	{attribute 'TcIecLibraryType'}
	{attribute 'external_name' := 'F_VN_HoughCircles_GUID_3208ACBE_0E75_B691_48A0_E9F1062BC23D'}
	(* Search for circles using the Hough transform. *)
	FUNCTION F_VN_HoughCircles : HRESULT
	VAR_INPUT
		ipSrcImage	:	ITcVnImage;	(* Source image (USINT, 1 channel, gray-level) *)
		ipCircles	:	REFERENCE TO ITcVnContainer;	(* Returns a container which is filled with the found circles (ContainerType_Vector_TcVnVector3_REAL; Each container element contains the x coordinate of the circle center [0], the y coordinate of the circle center [1], and the radius [2], respectively. Non-zero interface pointers are reused.) *)
		fInvAccuRatio	:	LREAL;	(* Inverted ratio of the accumulator size in relation to the source image's size (must be > 0. A value of 2 means that the size is halved in both directions.) *)
		fMinDist	:	LREAL;	(* Smallest allowed distance of two circles (must be > 0) *)
		hrPrev	:	HRESULT;	(* HRESULT indicating the result of previous operations (If SUCCEEDED(hrPrev) equals false, no operation is executed.) *)
	END_VAR

END_FUNCTION

// Functions/Image Analysis/Object Detection/F_VN_HoughCirclesExp

	{attribute 'TcIecLibraryType'}
	{attribute 'external_name' := 'F_VN_HoughCirclesExp_GUID_0524CE7C_E163_BD73_5710_38E608D89C08'}
	(* Search for circles using the Hough transform. (expert function) *)
	FUNCTION F_VN_HoughCirclesExp : HRESULT
	VAR_INPUT
		ipSrcImage	:	ITcVnImage;	(* Source image (USINT, 1 channel, gray-level) *)
		ipCircles	:	REFERENCE TO ITcVnContainer;	(* Returns a container which is filled with the found circles (ContainerType_Vector_TcVnVector3_REAL; Each container element contains the x coordinate of the circle center [0], the y coordinate of the circle center [1], and the radius [2], respectively. Non-zero interface pointers are reused.) *)
		fInvAccuRatio	:	LREAL;	(* Inverted ratio of the accumulator size in relation to the source image's size (must be > 0. A value of 2 means that the size is halved in both directions.) *)
		fMinDist	:	LREAL;	(* Smallest allowed distance of two circles (must be > 0) *)
		eHoughMethod	:	ETcVnHoughMethod;	(* Hough method to use (GRADIENT or GRADIENT_ALT) *)
		fParam1	:	LREAL;	(* First method specific parameter (GRADIENT, GRADIENT_ALT: upper threshold for canny edge detection, which must be > 0) *)
		fParam2	:	LREAL;	(* Second method specific parameter (GRADIENT: accumulator threshold for detecting circle centers, which must be > 0. GRADIENT_ALT: required circle perfectness, which must be > 0 and < 1, 1 would be a perfect circle) *)
		nMinRadius	:	UDINT;	(* Minimum circle radius allowed *)
		nMaxRadius	:	UDINT;	(* Maximum circle radius allowed (if 0, the value is internally set to max(image rows, image columns)) *)
		hrPrev	:	HRESULT;	(* HRESULT indicating the result of previous operations (If SUCCEEDED(hrPrev) equals false, no operation is executed.) *)
	END_VAR

END_FUNCTION

// Functions/Image Analysis/Object Detection/F_VN_HoughLines

	{attribute 'TcIecLibraryType'}
	{attribute 'external_name' := 'F_VN_HoughLines_GUID_82B94089_EA06_BA4D_5261_BCC69C56E98D'}
	(* Search for lines using the standard Hough transform. *)
	FUNCTION F_VN_HoughLines : HRESULT
	VAR_INPUT
		ipSrcImage	:	ITcVnImage;	(* Source image (USINT, 1 channel, binary, may be modified by the function) *)
		ipLines	:	REFERENCE TO ITcVnContainer;	(* Returns a container which is filled with the found lines (ContainerType_Vector_TcVnVector2_REAL; Each container element contains the distance from the origin [0] in pixels and the rotation angle [1] in radians, respectively. Non-zero interface pointers are reused.) *)
		fDistRes	:	LREAL;	(* Distance resolution of the accumulator (in pixels, must be > 0) *)
		fAngleRes	:	LREAL;	(* Angle resolution of the accumulator (in radians, must be > 0) *)
		nAccuThreshold	:	UDINT;	(* Accumulator threshold *)
		hrPrev	:	HRESULT;	(* HRESULT indicating the result of previous operations (If SUCCEEDED(hrPrev) equals false, no operation is executed.) *)
	END_VAR

END_FUNCTION

// Functions/Image Analysis/Object Detection/F_VN_HoughLinesExp

	{attribute 'TcIecLibraryType'}
	{attribute 'external_name' := 'F_VN_HoughLinesExp_GUID_A8676CC7_78FE_BBDF_4F0A_7E04EE46C3BD'}
	(* Search for lines using the standard Hough transform. (expert function) *)
	FUNCTION F_VN_HoughLinesExp : HRESULT
	VAR_INPUT
		ipSrcImage	:	ITcVnImage;	(* Source image (USINT, 1 channel, binary, may be modified by the function) *)
		ipLines	:	REFERENCE TO ITcVnContainer;	(* Returns a container which is filled with the found lines (ContainerType_Vector_TcVnVector2_REAL; Each container element contains the distance from the origin [0] in pixels and the rotation angle [1] in radians, respectively. Non-zero interface pointers are reused.) *)
		fDistRes	:	LREAL;	(* Distance resolution of the accumulator (in pixels, must be > 0) *)
		fAngleRes	:	LREAL;	(* Angle resolution of the accumulator (in radians, must be > 0) *)
		nAccuThreshold	:	UDINT;	(* Accumulator threshold *)
		fDistResDiv	:	LREAL;	(* Divisor of the distance resolution for the multi-scale Hough transform (>= 0, must be > 0 if fAngleResDiv is > 0) *)
		fAngleResDiv	:	LREAL;	(* Divisor of the angle resolution for the multi-scale Hough transform (>= 0, must be > 0 if fDistResDiv is > 0) *)
		hrPrev	:	HRESULT;	(* HRESULT indicating the result of previous operations (If SUCCEEDED(hrPrev) equals false, no operation is executed.) *)
	END_VAR

END_FUNCTION

// Functions/Image Analysis/Object Detection/F_VN_HoughLinesP

	{attribute 'TcIecLibraryType'}
	{attribute 'external_name' := 'F_VN_HoughLinesP_GUID_56A4DCAE_2908_B179_6CC2_F0080DB2F514'}
	(* Search for line segments using the probabilistic Hough transform. *)
	FUNCTION F_VN_HoughLinesP : HRESULT
	VAR_INPUT
		ipSrcImage	:	ITcVnImage;	(* Source image (USINT, 1 channel, binary, may be modified by the function) *)
		ipLines	:	REFERENCE TO ITcVnContainer;	(* Returns a container which is filled with the found line segments (ContainerType_Vector_TcVnVector4_DINT; Each container element contains the two ending points. Non-zero interface pointers are reused.) *)
		fDistRes	:	LREAL;	(* Distance resolution of the accumulator (in pixels, must be > 0) *)
		fAngleRes	:	LREAL;	(* Angle resolution of the accumulator (in radians, must be > 0) *)
		nAccuThreshold	:	UDINT;	(* Accumulator threshold *)
		hrPrev	:	HRESULT;	(* HRESULT indicating the result of previous operations (If SUCCEEDED(hrPrev) equals false, no operation is executed.) *)
	END_VAR

END_FUNCTION

// Functions/Image Analysis/Object Detection/F_VN_HoughLinesPExp

	{attribute 'TcIecLibraryType'}
	{attribute 'external_name' := 'F_VN_HoughLinesPExp_GUID_DBCDBAEB_C337_B034_483E_0DA75F1ED126'}
	(* Search for line segments using the probabilistic Hough transform. (expert function) *)
	FUNCTION F_VN_HoughLinesPExp : HRESULT
	VAR_INPUT
		ipSrcImage	:	ITcVnImage;	(* Source image (USINT, 1 channel, binary, may be modified by the function) *)
		ipLines	:	REFERENCE TO ITcVnContainer;	(* Returns a container which is filled with the found line segments (ContainerType_Vector_TcVnVector4_DINT; Each container element contains the two ending points. Non-zero interface pointers are reused.) *)
		fDistRes	:	LREAL;	(* Distance resolution of the accumulator (in pixels, must be > 0) *)
		fAngleRes	:	LREAL;	(* Angle resolution of the accumulator (in radians, must be > 0) *)
		nAccuThreshold	:	UDINT;	(* Accumulator threshold *)
		fMinLineLength	:	LREAL;	(* Minimum line length to search for *)
		fMaxLineGap	:	LREAL;	(* Maximum gap between points on the same line *)
		hrPrev	:	HRESULT;	(* HRESULT indicating the result of previous operations (If SUCCEEDED(hrPrev) equals false, no operation is executed.) *)
	END_VAR

END_FUNCTION

// Functions/Image Analysis/Object Detection/F_VN_MatchImageHuMoments

	{attribute 'TcIecLibraryType'}
	{attribute 'external_name' := 'F_VN_MatchImageHuMoments_GUID_658C7654_44DD_B199_410C_E15269A5A301'}
	(* Compare two images using the Hu moment invariants. *)
	FUNCTION F_VN_MatchImageHuMoments : HRESULT
	VAR_INPUT
		ipImage1	:	ITcVnImage;	(* First image (1 channel) *)
		ipImage2	:	ITcVnImage;	(* Second image (1 channel) *)
		eComparisonMethod	:	ETcVnContoursMatchComparisonMethod;	(* Method used for comparing the Hu moment invariants of the images *)
	END_VAR
	VAR_IN_OUT
		fDissimilarity	:	LREAL;	(* Returns the dissimilarity of the image Hu moment invariants depending on the chosen comparison method *)
	END_VAR
	VAR_INPUT
		hrPrev	:	HRESULT;	(* HRESULT indicating the result of previous operations (If SUCCEEDED(hrPrev) equals false, no operation is executed.) *)
	END_VAR

END_FUNCTION

// Functions/Image Analysis/Object Detection/F_VN_MatchTemplate

	{attribute 'TcIecLibraryType'}
	{attribute 'external_name' := 'F_VN_MatchTemplate_GUID_C0E3AE9A_E589_B4A4_40DE_437B35FB3E4E'}
	(* Match a template image with every location in the source image (using the TCVN_TMM_CCORR_NORMED method) and save the comparison results. *)
	FUNCTION F_VN_MatchTemplate : HRESULT
	VAR_INPUT
		ipSrcImage	:	ITcVnImage;	(* Source image (USINT or REAL, 1 or 3 channels) *)
		ipTemplateImage	:	ITcVnImage;	(* Template image (same type as ipSrcImage, smaller width and height) *)
		ipResultImage	:	REFERENCE TO ITcVnImage;	(* Returns the result image (REAL, normalized to [0..1], 1 channel, dimensions: (ipSrcImage.width - ipTemplateImage.width + 1) x (ipSrcImage.height - ipTemplateImage.height + 1). The best match is the global maximum. The position in ipResultImage is the top-left corner of ipTemplateImage position in ipSrcImage) *)
		hrPrev	:	HRESULT;	(* HRESULT indicating the result of previous operations (If SUCCEEDED(hrPrev) equals false, no operation is executed.) *)
	END_VAR

END_FUNCTION

// Functions/Image Analysis/Object Detection/F_VN_MatchTemplateExp

	{attribute 'TcIecLibraryType'}
	{attribute 'external_name' := 'F_VN_MatchTemplateExp_GUID_3688990C_CB5C_B619_7B29_C2927793ABF1'}
	(* Match a template image with every location in the source image and save the comparison results. (expert function) *)
	FUNCTION F_VN_MatchTemplateExp : HRESULT
	VAR_INPUT
		ipSrcImage	:	ITcVnImage;	(* Source image (USINT or REAL, 1 or 3 channels) *)
		ipTemplateImage	:	ITcVnImage;	(* Template image (same type as ipSrcImage, smaller width and height) *)
		ipResultImage	:	REFERENCE TO ITcVnImage;	(* Returns the result image (REAL, 1 channel, dimensions: (ipSrcImage.width - ipTemplateImage.width + 1) x (ipSrcImage.height - ipTemplateImage.height + 1). The best match is the global minimum (SQDIFF(_NORMED)) or maximum (CCORR(_NORMED), CCOEFF(_NORMED)). The position in ipResultImage is the top-left corner of ipTemplateImage position in ipSrcImage) *)
		eMatchMethod	:	ETcVnTemplateMatchMethod;	(* Specifies the template match method *)
		ipTemplateMask	:	ITcVnImage;	(* Optional mask for ipTemplateImage (same type and size as ipTemplateImage) *)
		hrPrev	:	HRESULT;	(* HRESULT indicating the result of previous operations (If SUCCEEDED(hrPrev) equals false, no operation is executed.) *)
	END_VAR

END_FUNCTION

// Functions/Image Analysis/Object Detection/F_VN_MatchTemplateAndEvaluate

	{attribute 'TcIecLibraryType'}
	{attribute 'external_name' := 'F_VN_MatchTemplateAndEvaluate_GUID_D49E239B_E98E_B6BB_418B_C7F76F8FBBDE'}
	(* Match a template image with every location in the source image (using the TCVN_TMM_CCORR_NORMED method) and evaluate the comparison results. Returns a sorted list of possible matches (best match first). *)
	FUNCTION F_VN_MatchTemplateAndEvaluate : HRESULT
	VAR_INPUT
		ipSrcImage	:	ITcVnImage;	(* Source image (USINT or REAL, 1 or 3 channels) *)
		ipTemplateImage	:	ITcVnImage;	(* Template image (same type as ipSrcImage, smaller width and height) *)
		ipMatches	:	REFERENCE TO ITcVnContainer;	(* Returns the matching positions (ContainerType_Vector_TcVnPoint2_DINT, where each element represents the top-left corner of ipTemplateImage) in ipSrcImage, sorted by relevance (best match first) *)
		fMatchThreshold	:	REAL;	(* Threshold to separate relevant from irrelevant matches (0..1, 1.0  would be a perfect match. To find a suitable value, you could evaluate some sample result images of F_VN_MatchTemplate.) *)
		hrPrev	:	HRESULT;	(* HRESULT indicating the result of previous operations (If SUCCEEDED(hrPrev) equals false, no operation is executed.) *)
	END_VAR

END_FUNCTION

// Functions/Image Analysis/Object Detection/F_VN_MatchTemplateAndEvaluateExp

	{attribute 'TcIecLibraryType'}
	{attribute 'external_name' := 'F_VN_MatchTemplateAndEvaluateExp_GUID_52774CC8_42BC_B4E1_7940_5C35FFE0176F'}
	(* Match a template image with every location in the source image and evaluate the comparison results. Returns a sorted list of possible matches (best match first). (expert function) *)
	FUNCTION F_VN_MatchTemplateAndEvaluateExp : HRESULT
	VAR_INPUT
		ipSrcImage	:	ITcVnImage;	(* Source image (USINT or REAL, 1 or 3 channels) *)
		ipTemplateImage	:	ITcVnImage;	(* Template image (same type as ipSrcImage, smaller width and height) *)
		ipMatches	:	REFERENCE TO ITcVnContainer;	(* Returns the matching positions (ContainerType_Vector_TcVnPoint2_DINT, where each element represents the top-left corner of ipTemplateImage) in ipSrcImage, sorted by relevance (best match first) *)
		fMatchThreshold	:	REAL;	(* Threshold to separate relevant from irrelevant matches (0..1 for NORMED methods, otherwise dependent on template size and content. To find a suitable value, you could evaluate some sample result images of F_VN_MatchTemplateExp.) *)
		eMatchMethod	:	ETcVnTemplateMatchMethod;	(* Specifies the template match method *)
		ipTemplateMask	:	ITcVnImage;	(* Optional mask for ipTemplateImage (same type and size as ipTemplateImage) *)
		fScaleFactor	:	REAL;	(* Factor (0..1] to reduce source and template image width and height for better performance (but less accuracy!) *)
		eInterpolationType	:	ETcVnInterpolationType;	(* Image resize interpolation type (only used if fScaleFactor != 1, TCVN_IT_BILINEAR recommended for most cases) *)
		ipMatchValues	:	REFERENCE TO ITcVnContainer;	(* Optionally returns the matching values (ContainerType_Vector_REAL, same size and sort order as ipMatches. Set to 0 if not required.) *)
		hrPrev	:	HRESULT;	(* HRESULT indicating the result of previous operations (If SUCCEEDED(hrPrev) equals false, no operation is executed.) *)
	END_VAR

END_FUNCTION

// Functions/Basic Container Operations/F_VN_AppendToContainer/F_VN_AppendToContainer_ITcVnContainer

	{attribute 'TcIecLibraryType'}
	{attribute 'external_name' := 'F_VN_AppendToContainer_ITcVnContainer_GUID_0871CEBE_66D6_B0B1_506F_1DCDB966BE0C'}
	(* Append a single element to a container or concatenate containers (if ipElement has the same typeId as ipContainer). *)
	FUNCTION F_VN_AppendToContainer_ITcVnContainer : HRESULT
	VAR_INPUT
		ipElement	:	ITcVnContainer;	(* Single element to append to ipContainer or container with several elements to be concatenated *)
		ipContainer	:	ITcVnContainer;	(* Container to which the element(s) will be appended *)
		hrPrev	:	HRESULT;	(* HRESULT indicating the result of previous operations (If SUCCEEDED(hrPrev) equals false, no operation is executed.) *)
	END_VAR

END_FUNCTION

// Functions/Basic Container Operations/F_VN_AppendToContainer/F_VN_AppendToContainer_ITcVnForwardIterator

	{attribute 'TcIecLibraryType'}
	{attribute 'external_name' := 'F_VN_AppendToContainer_ITcVnForwardIterator_GUID_68FE249C_FAB2_B211_7831_6890B9756309'}
	(* Append a single element (represented by an iterator)to a container. *)
	FUNCTION F_VN_AppendToContainer_ITcVnForwardIterator : HRESULT
	VAR_INPUT
		ipElement	:	ITcVnForwardIterator;	(* Single element to append to ipContainer *)
		ipContainer	:	ITcVnContainer;	(* Container to which the element(s) will be appended *)
		hrPrev	:	HRESULT;	(* HRESULT indicating the result of previous operations (If SUCCEEDED(hrPrev) equals false, no operation is executed.) *)
	END_VAR

END_FUNCTION

// Functions/Basic Container Operations/F_VN_AppendToContainer/F_VN_AppendToContainer_DINT

	{attribute 'TcIecLibraryType'}
	{attribute 'external_name' := 'F_VN_AppendToContainer_DINT_GUID_C5E3F485_1C44_B21C_61E3_958AE9652A0F'}
	(* Append a single element of type DINT to a container. *)
	FUNCTION F_VN_AppendToContainer_DINT : HRESULT
	VAR_INPUT
		nElement	:	DINT;	(* Single element to append to ipContainer *)
		ipContainer	:	ITcVnContainer;	(* Container to which the element will be appended *)
		hrPrev	:	HRESULT;	(* HRESULT indicating the result of previous operations (If SUCCEEDED(hrPrev) equals false, no operation is executed.) *)
	END_VAR

END_FUNCTION

// Functions/Basic Container Operations/F_VN_AppendToContainer/F_VN_AppendToContainer_INT

	{attribute 'TcIecLibraryType'}
	{attribute 'external_name' := 'F_VN_AppendToContainer_INT_GUID_1FA26B77_78C9_B37E_7C55_B9AB60A4781A'}
	(* Append a single element of type INT to a container. *)
	FUNCTION F_VN_AppendToContainer_INT : HRESULT
	VAR_INPUT
		nElement	:	INT;	(* Single element to append to ipContainer *)
		ipContainer	:	ITcVnContainer;	(* Container to which the element will be appended *)
		hrPrev	:	HRESULT;	(* HRESULT indicating the result of previous operations (If SUCCEEDED(hrPrev) equals false, no operation is executed.) *)
	END_VAR

END_FUNCTION

// Functions/Basic Container Operations/F_VN_AppendToContainer/F_VN_AppendToContainer_ITcVnImage

	{attribute 'TcIecLibraryType'}
	{attribute 'external_name' := 'F_VN_AppendToContainer_ITcVnImage_GUID_994AF0C6_0E53_B461_4DF2_1F839F8C5366'}
	(* Append a single element of type ITcVnImage to a container. *)
	FUNCTION F_VN_AppendToContainer_ITcVnImage : HRESULT
	VAR_INPUT
		ipElement	:	ITcVnImage;	(* Single element to append to ipContainer *)
		ipContainer	:	ITcVnContainer;	(* Container to which the element will be appended *)
		hrPrev	:	HRESULT;	(* HRESULT indicating the result of previous operations (If SUCCEEDED(hrPrev) equals false, no operation is executed.) *)
	END_VAR

END_FUNCTION

// Functions/Basic Container Operations/F_VN_AppendToContainer/F_VN_AppendToContainer_LREAL

	{attribute 'TcIecLibraryType'}
	{attribute 'external_name' := 'F_VN_AppendToContainer_LREAL_GUID_322EEAAD_BF59_BEC4_5462_10B3F9F43735'}
	(* Append a single element of type LREAL to a container. *)
	FUNCTION F_VN_AppendToContainer_LREAL : HRESULT
	VAR_INPUT
		fElement	:	LREAL;	(* Single element to append to ipContainer *)
		ipContainer	:	ITcVnContainer;	(* Container to which the element will be appended *)
		hrPrev	:	HRESULT;	(* HRESULT indicating the result of previous operations (If SUCCEEDED(hrPrev) equals false, no operation is executed.) *)
	END_VAR

END_FUNCTION

// Functions/Basic Container Operations/F_VN_AppendToContainer/F_VN_AppendToContainer_REAL

	{attribute 'TcIecLibraryType'}
	{attribute 'external_name' := 'F_VN_AppendToContainer_REAL_GUID_2B2B32F2_F49E_B830_4DE6_D5239ABAA89F'}
	(* Append a single element of type REAL to a container. *)
	FUNCTION F_VN_AppendToContainer_REAL : HRESULT
	VAR_INPUT
		fElement	:	REAL;	(* Single element to append to ipContainer *)
		ipContainer	:	ITcVnContainer;	(* Container to which the element will be appended *)
		hrPrev	:	HRESULT;	(* HRESULT indicating the result of previous operations (If SUCCEEDED(hrPrev) equals false, no operation is executed.) *)
	END_VAR

END_FUNCTION

// Functions/Basic Container Operations/F_VN_AppendToContainer/F_VN_AppendToContainer_SINT

	{attribute 'TcIecLibraryType'}
	{attribute 'external_name' := 'F_VN_AppendToContainer_SINT_GUID_AD0EA3F8_4615_B49A_4901_B8FA24011DED'}
	(* Append a single element of type SINT to a container. *)
	FUNCTION F_VN_AppendToContainer_SINT : HRESULT
	VAR_INPUT
		nElement	:	SINT;	(* Single element to append to ipContainer *)
		ipContainer	:	ITcVnContainer;	(* Container to which the element will be appended *)
		hrPrev	:	HRESULT;	(* HRESULT indicating the result of previous operations (If SUCCEEDED(hrPrev) equals false, no operation is executed.) *)
	END_VAR

END_FUNCTION

// Functions/Basic Container Operations/F_VN_AppendToContainer/F_VN_AppendToContainer_TcVnDMatch

	{attribute 'TcIecLibraryType'}
	{attribute 'external_name' := 'F_VN_AppendToContainer_TcVnDMatch_GUID_B7089787_0242_B315_4452_3A9278244513'}
	(* Append a single element of type TcVnDMatch to a container. *)
	FUNCTION F_VN_AppendToContainer_TcVnDMatch : HRESULT
	VAR_IN_OUT
		stElement	:	TcVnDMatch;	(* Single element to append to ipContainer *)
	END_VAR
	VAR_INPUT
		ipContainer	:	ITcVnContainer;	(* Container to which the element will be appended *)
		hrPrev	:	HRESULT;	(* HRESULT indicating the result of previous operations (If SUCCEEDED(hrPrev) equals false, no operation is executed.) *)
	END_VAR

END_FUNCTION

// Functions/Basic Container Operations/F_VN_AppendToContainer/F_VN_AppendToContainer_TcVnKeyPoint

	{attribute 'TcIecLibraryType'}
	{attribute 'external_name' := 'F_VN_AppendToContainer_TcVnKeyPoint_GUID_5E909463_2C7F_B636_51C1_80D41999F1FF'}
	(* Append a single element of type TcVnKeyPoint to a container. *)
	FUNCTION F_VN_AppendToContainer_TcVnKeyPoint : HRESULT
	VAR_IN_OUT
		stElement	:	TcVnKeyPoint;	(* Single element to append to ipContainer *)
	END_VAR
	VAR_INPUT
		ipContainer	:	ITcVnContainer;	(* Container to which the element will be appended *)
		hrPrev	:	HRESULT;	(* HRESULT indicating the result of previous operations (If SUCCEEDED(hrPrev) equals false, no operation is executed.) *)
	END_VAR

END_FUNCTION

// Functions/Basic Container Operations/F_VN_AppendToContainer/F_VN_AppendToContainer_TcVnPoint2_DINT

	{attribute 'TcIecLibraryType'}
	{attribute 'external_name' := 'F_VN_AppendToContainer_TcVnPoint2_DINT_GUID_61BA2EFB_B8BC_BFA0_630E_75DD36BF3AF5'}
	(* Append a single element of type TcVnPoint2_DINT to a container. *)
	FUNCTION F_VN_AppendToContainer_TcVnPoint2_DINT : HRESULT
	VAR_IN_OUT
		aElement	:	TcVnPoint2_DINT;	(* Single element to append to ipContainer *)
	END_VAR
	VAR_INPUT
		ipContainer	:	ITcVnContainer;	(* Container to which the element will be appended *)
		hrPrev	:	HRESULT;	(* HRESULT indicating the result of previous operations (If SUCCEEDED(hrPrev) equals false, no operation is executed.) *)
	END_VAR

END_FUNCTION

// Functions/Basic Container Operations/F_VN_AppendToContainer/F_VN_AppendToContainer_TcVnPoint2_LREAL

	{attribute 'TcIecLibraryType'}
	{attribute 'external_name' := 'F_VN_AppendToContainer_TcVnPoint2_LREAL_GUID_9578CCDD_C312_B676_7B95_A36643CB113E'}
	(* Append a single element of type TcVnPoint2_LREAL to a container. *)
	FUNCTION F_VN_AppendToContainer_TcVnPoint2_LREAL : HRESULT
	VAR_IN_OUT
		aElement	:	TcVnPoint2_LREAL;	(* Single element to append to ipContainer *)
	END_VAR
	VAR_INPUT
		ipContainer	:	ITcVnContainer;	(* Container to which the element will be appended *)
		hrPrev	:	HRESULT;	(* HRESULT indicating the result of previous operations (If SUCCEEDED(hrPrev) equals false, no operation is executed.) *)
	END_VAR

END_FUNCTION

// Functions/Basic Container Operations/F_VN_AppendToContainer/F_VN_AppendToContainer_TcVnPoint2_REAL

	{attribute 'TcIecLibraryType'}
	{attribute 'external_name' := 'F_VN_AppendToContainer_TcVnPoint2_REAL_GUID_2CACAC7F_BF8B_B238_50E3_05B26FF81174'}
	(* Append a single element of type TcVnPoint2_REAL to a container. *)
	FUNCTION F_VN_AppendToContainer_TcVnPoint2_REAL : HRESULT
	VAR_IN_OUT
		aElement	:	TcVnPoint2_REAL;	(* Single element to append to ipContainer *)
	END_VAR
	VAR_INPUT
		ipContainer	:	ITcVnContainer;	(* Container to which the element will be appended *)
		hrPrev	:	HRESULT;	(* HRESULT indicating the result of previous operations (If SUCCEEDED(hrPrev) equals false, no operation is executed.) *)
	END_VAR

END_FUNCTION

// Functions/Basic Container Operations/F_VN_AppendToContainer/F_VN_AppendToContainer_TcVnPoint3_LREAL

	{attribute 'TcIecLibraryType'}
	{attribute 'external_name' := 'F_VN_AppendToContainer_TcVnPoint3_LREAL_GUID_C00DAD65_4FEA_B107_711B_0C106CCBB85A'}
	(* Append a single element of type TcVnPoint3_LREAL to a container. *)
	FUNCTION F_VN_AppendToContainer_TcVnPoint3_LREAL : HRESULT
	VAR_IN_OUT
		aElement	:	TcVnPoint3_LREAL;	(* Single element to append to ipContainer *)
	END_VAR
	VAR_INPUT
		ipContainer	:	ITcVnContainer;	(* Container to which the element will be appended *)
		hrPrev	:	HRESULT;	(* HRESULT indicating the result of previous operations (If SUCCEEDED(hrPrev) equals false, no operation is executed.) *)
	END_VAR

END_FUNCTION

// Functions/Basic Container Operations/F_VN_AppendToContainer/F_VN_AppendToContainer_TcVnPoint3_REAL

	{attribute 'TcIecLibraryType'}
	{attribute 'external_name' := 'F_VN_AppendToContainer_TcVnPoint3_REAL_GUID_DCD53F51_0FDB_B6B9_6DCB_4B5117963B6D'}
	(* Append a single element of type TcVnPoint3_REAL to a container. *)
	FUNCTION F_VN_AppendToContainer_TcVnPoint3_REAL : HRESULT
	VAR_IN_OUT
		aElement	:	TcVnPoint3_REAL;	(* Single element to append to ipContainer *)
	END_VAR
	VAR_INPUT
		ipContainer	:	ITcVnContainer;	(* Container to which the element will be appended *)
		hrPrev	:	HRESULT;	(* HRESULT indicating the result of previous operations (If SUCCEEDED(hrPrev) equals false, no operation is executed.) *)
	END_VAR

END_FUNCTION

// Functions/Basic Container Operations/F_VN_AppendToContainer/F_VN_AppendToContainer_TcVnRectangle_DINT

	{attribute 'TcIecLibraryType'}
	{attribute 'external_name' := 'F_VN_AppendToContainer_TcVnRectangle_DINT_GUID_C4A818BF_201D_B4FB_7B4B_564F3F6D47CE'}
	(* Append a single element of type TcVnRectangle_DINT to a container. *)
	FUNCTION F_VN_AppendToContainer_TcVnRectangle_DINT : HRESULT
	VAR_IN_OUT
		stElement	:	TcVnRectangle_DINT;	(* Single element to append to ipContainer *)
	END_VAR
	VAR_INPUT
		ipContainer	:	ITcVnContainer;	(* Container to which the element will be appended *)
		hrPrev	:	HRESULT;	(* HRESULT indicating the result of previous operations (If SUCCEEDED(hrPrev) equals false, no operation is executed.) *)
	END_VAR

END_FUNCTION

// Functions/Basic Container Operations/F_VN_AppendToContainer/F_VN_AppendToContainer_TcVnVector2_DINT

	{attribute 'TcIecLibraryType'}
	{attribute 'external_name' := 'F_VN_AppendToContainer_TcVnVector2_DINT_GUID_41B34E71_A627_B579_4E88_D7D74BBEB1E5'}
	(* Append a single element of type TcVnVector2_DINT to a container. *)
	FUNCTION F_VN_AppendToContainer_TcVnVector2_DINT : HRESULT
	VAR_IN_OUT
		aElement	:	TcVnVector2_DINT;	(* Single element to append to ipContainer *)
	END_VAR
	VAR_INPUT
		ipContainer	:	ITcVnContainer;	(* Container to which the element will be appended *)
		hrPrev	:	HRESULT;	(* HRESULT indicating the result of previous operations (If SUCCEEDED(hrPrev) equals false, no operation is executed.) *)
	END_VAR

END_FUNCTION

// Functions/Basic Container Operations/F_VN_AppendToContainer/F_VN_AppendToContainer_TcVnVector2_INT

	{attribute 'TcIecLibraryType'}
	{attribute 'external_name' := 'F_VN_AppendToContainer_TcVnVector2_INT_GUID_03190075_1655_BB8D_5670_7DFA56918C83'}
	(* Append a single element of type TcVnVector2_INT to a container. *)
	FUNCTION F_VN_AppendToContainer_TcVnVector2_INT : HRESULT
	VAR_IN_OUT
		aElement	:	TcVnVector2_INT;	(* Single element to append to ipContainer *)
	END_VAR
	VAR_INPUT
		ipContainer	:	ITcVnContainer;	(* Container to which the element will be appended *)
		hrPrev	:	HRESULT;	(* HRESULT indicating the result of previous operations (If SUCCEEDED(hrPrev) equals false, no operation is executed.) *)
	END_VAR

END_FUNCTION

// Functions/Basic Container Operations/F_VN_AppendToContainer/F_VN_AppendToContainer_TcVnVector2_REAL

	{attribute 'TcIecLibraryType'}
	{attribute 'external_name' := 'F_VN_AppendToContainer_TcVnVector2_REAL_GUID_CAA9172F_D581_B4EB_508B_C992A7AC72E9'}
	(* Append a single element of type TcVnVector2_REAL to a container. *)
	FUNCTION F_VN_AppendToContainer_TcVnVector2_REAL : HRESULT
	VAR_IN_OUT
		aElement	:	TcVnVector2_REAL;	(* Single element to append to ipContainer *)
	END_VAR
	VAR_INPUT
		ipContainer	:	ITcVnContainer;	(* Container to which the element will be appended *)
		hrPrev	:	HRESULT;	(* HRESULT indicating the result of previous operations (If SUCCEEDED(hrPrev) equals false, no operation is executed.) *)
	END_VAR

END_FUNCTION

// Functions/Basic Container Operations/F_VN_AppendToContainer/F_VN_AppendToContainer_TcVnVector2_SINT

	{attribute 'TcIecLibraryType'}
	{attribute 'external_name' := 'F_VN_AppendToContainer_TcVnVector2_SINT_GUID_B243487F_92C1_BF7E_71E2_97E88C51A164'}
	(* Append a single element of type TcVnVector2_SINT to a container. *)
	FUNCTION F_VN_AppendToContainer_TcVnVector2_SINT : HRESULT
	VAR_IN_OUT
		aElement	:	TcVnVector2_SINT;	(* Single element to append to ipContainer *)
	END_VAR
	VAR_INPUT
		ipContainer	:	ITcVnContainer;	(* Container to which the element will be appended *)
		hrPrev	:	HRESULT;	(* HRESULT indicating the result of previous operations (If SUCCEEDED(hrPrev) equals false, no operation is executed.) *)
	END_VAR

END_FUNCTION

// Functions/Basic Container Operations/F_VN_AppendToContainer/F_VN_AppendToContainer_TcVnVector2_UINT

	{attribute 'TcIecLibraryType'}
	{attribute 'external_name' := 'F_VN_AppendToContainer_TcVnVector2_UINT_GUID_65CA8312_34CD_BCB3_4316_349611E62963'}
	(* Append a single element of type TcVnVector2_UINT to a container. *)
	FUNCTION F_VN_AppendToContainer_TcVnVector2_UINT : HRESULT
	VAR_IN_OUT
		aElement	:	TcVnVector2_UINT;	(* Single element to append to ipContainer *)
	END_VAR
	VAR_INPUT
		ipContainer	:	ITcVnContainer;	(* Container to which the element will be appended *)
		hrPrev	:	HRESULT;	(* HRESULT indicating the result of previous operations (If SUCCEEDED(hrPrev) equals false, no operation is executed.) *)
	END_VAR

END_FUNCTION

// Functions/Basic Container Operations/F_VN_AppendToContainer/F_VN_AppendToContainer_TcVnVector2_USINT

	{attribute 'TcIecLibraryType'}
	{attribute 'external_name' := 'F_VN_AppendToContainer_TcVnVector2_USINT_GUID_CFDE5759_AA22_BAFD_4045_17761752DF7A'}
	(* Append a single element of type TcVnVector2_USINT to a container. *)
	FUNCTION F_VN_AppendToContainer_TcVnVector2_USINT : HRESULT
	VAR_IN_OUT
		aElement	:	TcVnVector2_USINT;	(* Single element to append to ipContainer *)
	END_VAR
	VAR_INPUT
		ipContainer	:	ITcVnContainer;	(* Container to which the element will be appended *)
		hrPrev	:	HRESULT;	(* HRESULT indicating the result of previous operations (If SUCCEEDED(hrPrev) equals false, no operation is executed.) *)
	END_VAR

END_FUNCTION

// Functions/Basic Container Operations/F_VN_AppendToContainer/F_VN_AppendToContainer_TcVnVector3_INT

	{attribute 'TcIecLibraryType'}
	{attribute 'external_name' := 'F_VN_AppendToContainer_TcVnVector3_INT_GUID_865E49A2_C2A9_B29E_4549_0BC3152D1033'}
	(* Append a single element of type TcVnVector3_INT to a container. *)
	FUNCTION F_VN_AppendToContainer_TcVnVector3_INT : HRESULT
	VAR_IN_OUT
		aElement	:	TcVnVector3_INT;	(* Single element to append to ipContainer *)
	END_VAR
	VAR_INPUT
		ipContainer	:	ITcVnContainer;	(* Container to which the element will be appended *)
		hrPrev	:	HRESULT;	(* HRESULT indicating the result of previous operations (If SUCCEEDED(hrPrev) equals false, no operation is executed.) *)
	END_VAR

END_FUNCTION

// Functions/Basic Container Operations/F_VN_AppendToContainer/F_VN_AppendToContainer_TcVnVector3_REAL

	{attribute 'TcIecLibraryType'}
	{attribute 'external_name' := 'F_VN_AppendToContainer_TcVnVector3_REAL_GUID_D2CCFE6F_59DD_B2C5_60F3_EB5A1DCAE86F'}
	(* Append a single element of type TcVnVector3_REAL to a container. *)
	FUNCTION F_VN_AppendToContainer_TcVnVector3_REAL : HRESULT
	VAR_IN_OUT
		aElement	:	TcVnVector3_REAL;	(* Single element to append to ipContainer *)
	END_VAR
	VAR_INPUT
		ipContainer	:	ITcVnContainer;	(* Container to which the element will be appended *)
		hrPrev	:	HRESULT;	(* HRESULT indicating the result of previous operations (If SUCCEEDED(hrPrev) equals false, no operation is executed.) *)
	END_VAR

END_FUNCTION

// Functions/Basic Container Operations/F_VN_AppendToContainer/F_VN_AppendToContainer_TcVnVector3_SINT

	{attribute 'TcIecLibraryType'}
	{attribute 'external_name' := 'F_VN_AppendToContainer_TcVnVector3_SINT_GUID_C0B410A5_2EC6_B0F0_49B3_B07241C8F6DE'}
	(* Append a single element of type TcVnVector3_SINT to a container. *)
	FUNCTION F_VN_AppendToContainer_TcVnVector3_SINT : HRESULT
	VAR_IN_OUT
		aElement	:	TcVnVector3_SINT;	(* Single element to append to ipContainer *)
	END_VAR
	VAR_INPUT
		ipContainer	:	ITcVnContainer;	(* Container to which the element will be appended *)
		hrPrev	:	HRESULT;	(* HRESULT indicating the result of previous operations (If SUCCEEDED(hrPrev) equals false, no operation is executed.) *)
	END_VAR

END_FUNCTION

// Functions/Basic Container Operations/F_VN_AppendToContainer/F_VN_AppendToContainer_TcVnVector3_UINT

	{attribute 'TcIecLibraryType'}
	{attribute 'external_name' := 'F_VN_AppendToContainer_TcVnVector3_UINT_GUID_F6024E8E_E5FB_BD9D_7C19_F5DA416AACF1'}
	(* Append a single element of type TcVnVector3_UINT to a container. *)
	FUNCTION F_VN_AppendToContainer_TcVnVector3_UINT : HRESULT
	VAR_IN_OUT
		aElement	:	TcVnVector3_UINT;	(* Single element to append to ipContainer *)
	END_VAR
	VAR_INPUT
		ipContainer	:	ITcVnContainer;	(* Container to which the element will be appended *)
		hrPrev	:	HRESULT;	(* HRESULT indicating the result of previous operations (If SUCCEEDED(hrPrev) equals false, no operation is executed.) *)
	END_VAR

END_FUNCTION

// Functions/Basic Container Operations/F_VN_AppendToContainer/F_VN_AppendToContainer_TcVnVector3_USINT

	{attribute 'TcIecLibraryType'}
	{attribute 'external_name' := 'F_VN_AppendToContainer_TcVnVector3_USINT_GUID_8B62F65E_08EA_B240_504E_B61CBAA0D91D'}
	(* Append a single element of type TcVnVector3_USINT to a container. *)
	FUNCTION F_VN_AppendToContainer_TcVnVector3_USINT : HRESULT
	VAR_IN_OUT
		aElement	:	TcVnVector3_USINT;	(* Single element to append to ipContainer *)
	END_VAR
	VAR_INPUT
		ipContainer	:	ITcVnContainer;	(* Container to which the element will be appended *)
		hrPrev	:	HRESULT;	(* HRESULT indicating the result of previous operations (If SUCCEEDED(hrPrev) equals false, no operation is executed.) *)
	END_VAR

END_FUNCTION

// Functions/Basic Container Operations/F_VN_AppendToContainer/F_VN_AppendToContainer_TcVnVector4_DINT

	{attribute 'TcIecLibraryType'}
	{attribute 'external_name' := 'F_VN_AppendToContainer_TcVnVector4_DINT_GUID_8BB3E3FF_2F4E_BC73_4B23_6733ABEE0780'}
	(* Append a single element of type TcVnVector4_DINT to a container. *)
	FUNCTION F_VN_AppendToContainer_TcVnVector4_DINT : HRESULT
	VAR_IN_OUT
		aElement	:	TcVnVector4_DINT;	(* Single element to append to ipContainer *)
	END_VAR
	VAR_INPUT
		ipContainer	:	ITcVnContainer;	(* Container to which the element will be appended *)
		hrPrev	:	HRESULT;	(* HRESULT indicating the result of previous operations (If SUCCEEDED(hrPrev) equals false, no operation is executed.) *)
	END_VAR

END_FUNCTION

// Functions/Basic Container Operations/F_VN_AppendToContainer/F_VN_AppendToContainer_TcVnVector4_INT

	{attribute 'TcIecLibraryType'}
	{attribute 'external_name' := 'F_VN_AppendToContainer_TcVnVector4_INT_GUID_80AE1EA5_7A7E_B9B0_4985_BB5D32954B0E'}
	(* Append a single element of type TcVnVector4_INT to a container. *)
	FUNCTION F_VN_AppendToContainer_TcVnVector4_INT : HRESULT
	VAR_IN_OUT
		aElement	:	TcVnVector4_INT;	(* Single element to append to ipContainer *)
	END_VAR
	VAR_INPUT
		ipContainer	:	ITcVnContainer;	(* Container to which the element will be appended *)
		hrPrev	:	HRESULT;	(* HRESULT indicating the result of previous operations (If SUCCEEDED(hrPrev) equals false, no operation is executed.) *)
	END_VAR

END_FUNCTION

// Functions/Basic Container Operations/F_VN_AppendToContainer/F_VN_AppendToContainer_TcVnVector4_LREAL

	{attribute 'TcIecLibraryType'}
	{attribute 'external_name' := 'F_VN_AppendToContainer_TcVnVector4_LREAL_GUID_EB913DE2_DA93_BA7B_473D_8239404B5042'}
	(* Append a single element of type TcVnVector4_LREAL to a container. *)
	FUNCTION F_VN_AppendToContainer_TcVnVector4_LREAL : HRESULT
	VAR_IN_OUT
		aElement	:	TcVnVector4_LREAL;	(* Single element to append to ipContainer *)
	END_VAR
	VAR_INPUT
		ipContainer	:	ITcVnContainer;	(* Container to which the element will be appended *)
		hrPrev	:	HRESULT;	(* HRESULT indicating the result of previous operations (If SUCCEEDED(hrPrev) equals false, no operation is executed.) *)
	END_VAR

END_FUNCTION

// Functions/Basic Container Operations/F_VN_AppendToContainer/F_VN_AppendToContainer_TcVnVector4_SINT

	{attribute 'TcIecLibraryType'}
	{attribute 'external_name' := 'F_VN_AppendToContainer_TcVnVector4_SINT_GUID_0C452B4A_D316_B59E_437F_F319934F215D'}
	(* Append a single element of type TcVnVector4_SINT to a container. *)
	FUNCTION F_VN_AppendToContainer_TcVnVector4_SINT : HRESULT
	VAR_IN_OUT
		aElement	:	TcVnVector4_SINT;	(* Single element to append to ipContainer *)
	END_VAR
	VAR_INPUT
		ipContainer	:	ITcVnContainer;	(* Container to which the element will be appended *)
		hrPrev	:	HRESULT;	(* HRESULT indicating the result of previous operations (If SUCCEEDED(hrPrev) equals false, no operation is executed.) *)
	END_VAR

END_FUNCTION

// Functions/Basic Container Operations/F_VN_AppendToContainer/F_VN_AppendToContainer_TcVnVector4_UINT

	{attribute 'TcIecLibraryType'}
	{attribute 'external_name' := 'F_VN_AppendToContainer_TcVnVector4_UINT_GUID_0032CD21_D254_B26C_7A07_E6D6874AB4CC'}
	(* Append a single element of type TcVnVector4_UINT to a container. *)
	FUNCTION F_VN_AppendToContainer_TcVnVector4_UINT : HRESULT
	VAR_IN_OUT
		aElement	:	TcVnVector4_UINT;	(* Single element to append to ipContainer *)
	END_VAR
	VAR_INPUT
		ipContainer	:	ITcVnContainer;	(* Container to which the element will be appended *)
		hrPrev	:	HRESULT;	(* HRESULT indicating the result of previous operations (If SUCCEEDED(hrPrev) equals false, no operation is executed.) *)
	END_VAR

END_FUNCTION

// Functions/Basic Container Operations/F_VN_AppendToContainer/F_VN_AppendToContainer_TcVnVector4_USINT

	{attribute 'TcIecLibraryType'}
	{attribute 'external_name' := 'F_VN_AppendToContainer_TcVnVector4_USINT_GUID_EC0B014C_363A_BF2F_6D81_097AF29A2E32'}
	(* Append a single element of type TcVnVector4_USINT to a container. *)
	FUNCTION F_VN_AppendToContainer_TcVnVector4_USINT : HRESULT
	VAR_IN_OUT
		aElement	:	TcVnVector4_USINT;	(* Single element to append to ipContainer *)
	END_VAR
	VAR_INPUT
		ipContainer	:	ITcVnContainer;	(* Container to which the element will be appended *)
		hrPrev	:	HRESULT;	(* HRESULT indicating the result of previous operations (If SUCCEEDED(hrPrev) equals false, no operation is executed.) *)
	END_VAR

END_FUNCTION

// Functions/Basic Container Operations/F_VN_AppendToContainer/F_VN_AppendToContainer_UDINT

	{attribute 'TcIecLibraryType'}
	{attribute 'external_name' := 'F_VN_AppendToContainer_UDINT_GUID_07FC158B_CFC8_B0A5_770B_691D25F2923E'}
	(* Append a single element of type UDINT to a container. *)
	FUNCTION F_VN_AppendToContainer_UDINT : HRESULT
	VAR_INPUT
		nElement	:	UDINT;	(* Single element to append to ipContainer *)
		ipContainer	:	ITcVnContainer;	(* Container to which the element will be appended *)
		hrPrev	:	HRESULT;	(* HRESULT indicating the result of previous operations (If SUCCEEDED(hrPrev) equals false, no operation is executed.) *)
	END_VAR

END_FUNCTION

// Functions/Basic Container Operations/F_VN_AppendToContainer/F_VN_AppendToContainer_UINT

	{attribute 'TcIecLibraryType'}
	{attribute 'external_name' := 'F_VN_AppendToContainer_UINT_GUID_BDB75763_84AF_B740_41A9_314125C5A350'}
	(* Append a single element of type UINT to a container. *)
	FUNCTION F_VN_AppendToContainer_UINT : HRESULT
	VAR_INPUT
		nElement	:	UINT;	(* Single element to append to ipContainer *)
		ipContainer	:	ITcVnContainer;	(* Container to which the element will be appended *)
		hrPrev	:	HRESULT;	(* HRESULT indicating the result of previous operations (If SUCCEEDED(hrPrev) equals false, no operation is executed.) *)
	END_VAR

END_FUNCTION

// Functions/Basic Container Operations/F_VN_AppendToContainer/F_VN_AppendToContainer_ULINT

	{attribute 'TcIecLibraryType'}
	{attribute 'external_name' := 'F_VN_AppendToContainer_ULINT_GUID_31AA49B0_A8DE_B40B_4286_64C865B39163'}
	(* Append a single element of type ULINT to a container. *)
	FUNCTION F_VN_AppendToContainer_ULINT : HRESULT
	VAR_INPUT
		nElement	:	ULINT;	(* Single element to append to ipContainer *)
		ipContainer	:	ITcVnContainer;	(* Container to which the element will be appended *)
		hrPrev	:	HRESULT;	(* HRESULT indicating the result of previous operations (If SUCCEEDED(hrPrev) equals false, no operation is executed.) *)
	END_VAR

END_FUNCTION

// Functions/Basic Container Operations/F_VN_AppendToContainer/F_VN_AppendToContainer_USINT

	{attribute 'TcIecLibraryType'}
	{attribute 'external_name' := 'F_VN_AppendToContainer_USINT_GUID_8F2D6821_4D5B_B313_5DEE_BB4B65282616'}
	(* Append a single element of type USINT to a container. *)
	FUNCTION F_VN_AppendToContainer_USINT : HRESULT
	VAR_INPUT
		nElement	:	USINT;	(* Single element to append to ipContainer *)
		ipContainer	:	ITcVnContainer;	(* Container to which the element will be appended *)
		hrPrev	:	HRESULT;	(* HRESULT indicating the result of previous operations (If SUCCEEDED(hrPrev) equals false, no operation is executed.) *)
	END_VAR

END_FUNCTION

// Functions/Basic Container Operations/F_VN_FillContainer/F_VN_FillContainer_DINT

	{attribute 'TcIecLibraryType'}
	{attribute 'external_name' := 'F_VN_FillContainer_DINT_GUID_8BB266DC_9DD3_B627_565F_7067D41D7538'}
	(* Fill the container with the specified value. Only possible for containers with basic elements. *)
	FUNCTION F_VN_FillContainer_DINT : HRESULT
	VAR_INPUT
		ipContainer	:	ITcVnContainer;	(* Container with basic elements *)
		nValue	:	DINT;	(* Value to set the container elements *)
		hrPrev	:	HRESULT;	(* HRESULT indicating the result of previous operations (If SUCCEEDED(hrPrev) equals false, no operation is executed.) *)
	END_VAR

END_FUNCTION

// Functions/Basic Container Operations/F_VN_FillContainer/F_VN_FillContainer_INT

	{attribute 'TcIecLibraryType'}
	{attribute 'external_name' := 'F_VN_FillContainer_INT_GUID_0D5FEBDD_6399_B344_4F23_559608459CC7'}
	(* Fill the container with the specified value. Only possible for containers with basic elements. *)
	FUNCTION F_VN_FillContainer_INT : HRESULT
	VAR_INPUT
		ipContainer	:	ITcVnContainer;	(* Container with basic elements *)
		nValue	:	INT;	(* Value to set the container elements *)
		hrPrev	:	HRESULT;	(* HRESULT indicating the result of previous operations (If SUCCEEDED(hrPrev) equals false, no operation is executed.) *)
	END_VAR

END_FUNCTION

// Functions/Basic Container Operations/F_VN_FillContainer/F_VN_FillContainer_ITcVnImage

	{attribute 'TcIecLibraryType'}
	{attribute 'external_name' := 'F_VN_FillContainer_ITcVnImage_GUID_A1258E31_3B81_BA73_614D_90858A512D0D'}
	(* Fill the container with the specified value. Only possible for containers with basic elements. *)
	FUNCTION F_VN_FillContainer_ITcVnImage : HRESULT
	VAR_INPUT
		ipContainer	:	ITcVnContainer;	(* Container with basic elements *)
		ipValue	:	ITcVnImage;	(* Value to set the container elements *)
		hrPrev	:	HRESULT;	(* HRESULT indicating the result of previous operations (If SUCCEEDED(hrPrev) equals false, no operation is executed.) *)
	END_VAR

END_FUNCTION

// Functions/Basic Container Operations/F_VN_FillContainer/F_VN_FillContainer_LREAL

	{attribute 'TcIecLibraryType'}
	{attribute 'external_name' := 'F_VN_FillContainer_LREAL_GUID_0EB3FA1D_6B4E_B9F9_57FC_0DED14EB922F'}
	(* Fill the container with the specified value. Only possible for containers with basic elements. *)
	FUNCTION F_VN_FillContainer_LREAL : HRESULT
	VAR_INPUT
		ipContainer	:	ITcVnContainer;	(* Container with basic elements *)
		fValue	:	LREAL;	(* Value to set the container elements *)
		hrPrev	:	HRESULT;	(* HRESULT indicating the result of previous operations (If SUCCEEDED(hrPrev) equals false, no operation is executed.) *)
	END_VAR

END_FUNCTION

// Functions/Basic Container Operations/F_VN_FillContainer/F_VN_FillContainer_REAL

	{attribute 'TcIecLibraryType'}
	{attribute 'external_name' := 'F_VN_FillContainer_REAL_GUID_53B9D44F_7269_B320_6944_9E8CB7215B15'}
	(* Fill the container with the specified value. Only possible for containers with basic elements. *)
	FUNCTION F_VN_FillContainer_REAL : HRESULT
	VAR_INPUT
		ipContainer	:	ITcVnContainer;	(* Container with basic elements *)
		fValue	:	REAL;	(* Value to set the container elements *)
		hrPrev	:	HRESULT;	(* HRESULT indicating the result of previous operations (If SUCCEEDED(hrPrev) equals false, no operation is executed.) *)
	END_VAR

END_FUNCTION

// Functions/Basic Container Operations/F_VN_FillContainer/F_VN_FillContainer_SINT

	{attribute 'TcIecLibraryType'}
	{attribute 'external_name' := 'F_VN_FillContainer_SINT_GUID_74859358_058A_B104_5BCB_AD33D56BA120'}
	(* Fill the container with the specified value. Only possible for containers with basic elements. *)
	FUNCTION F_VN_FillContainer_SINT : HRESULT
	VAR_INPUT
		ipContainer	:	ITcVnContainer;	(* Container with basic elements *)
		nValue	:	SINT;	(* Value to set the container elements *)
		hrPrev	:	HRESULT;	(* HRESULT indicating the result of previous operations (If SUCCEEDED(hrPrev) equals false, no operation is executed.) *)
	END_VAR

END_FUNCTION

// Functions/Basic Container Operations/F_VN_FillContainer/F_VN_FillContainer_TcVnDMatch

	{attribute 'TcIecLibraryType'}
	{attribute 'external_name' := 'F_VN_FillContainer_TcVnDMatch_GUID_1945276A_7A89_B552_5CEE_6CF2E817D3E8'}
	(* Fill the container with the specified value. Only possible for containers with basic elements. *)
	FUNCTION F_VN_FillContainer_TcVnDMatch : HRESULT
	VAR_INPUT
		ipContainer	:	ITcVnContainer;	(* Container with basic elements *)
	END_VAR
	VAR_IN_OUT
		stValue	:	TcVnDMatch;	(* Value to set the container elements *)
	END_VAR
	VAR_INPUT
		hrPrev	:	HRESULT;	(* HRESULT indicating the result of previous operations (If SUCCEEDED(hrPrev) equals false, no operation is executed.) *)
	END_VAR

END_FUNCTION

// Functions/Basic Container Operations/F_VN_FillContainer/F_VN_FillContainer_TcVnKeyPoint

	{attribute 'TcIecLibraryType'}
	{attribute 'external_name' := 'F_VN_FillContainer_TcVnKeyPoint_GUID_93F5697E_0406_B001_550F_074DFB818BFF'}
	(* Fill the container with the specified value. Only possible for containers with basic elements. *)
	FUNCTION F_VN_FillContainer_TcVnKeyPoint : HRESULT
	VAR_INPUT
		ipContainer	:	ITcVnContainer;	(* Container with basic elements *)
	END_VAR
	VAR_IN_OUT
		stValue	:	TcVnKeyPoint;	(* Value to set the container elements *)
	END_VAR
	VAR_INPUT
		hrPrev	:	HRESULT;	(* HRESULT indicating the result of previous operations (If SUCCEEDED(hrPrev) equals false, no operation is executed.) *)
	END_VAR

END_FUNCTION

// Functions/Basic Container Operations/F_VN_FillContainer/F_VN_FillContainer_TcVnPoint2_DINT

	{attribute 'TcIecLibraryType'}
	{attribute 'external_name' := 'F_VN_FillContainer_TcVnPoint2_DINT_GUID_896AA622_F81D_B871_5AC2_A56F3E0FE41E'}
	(* Fill the container with the specified value. Only possible for containers with basic elements. *)
	FUNCTION F_VN_FillContainer_TcVnPoint2_DINT : HRESULT
	VAR_INPUT
		ipContainer	:	ITcVnContainer;	(* Container with basic elements *)
	END_VAR
	VAR_IN_OUT
		aValue	:	TcVnPoint2_DINT;	(* Value to set the container elements *)
	END_VAR
	VAR_INPUT
		hrPrev	:	HRESULT;	(* HRESULT indicating the result of previous operations (If SUCCEEDED(hrPrev) equals false, no operation is executed.) *)
	END_VAR

END_FUNCTION

// Functions/Basic Container Operations/F_VN_FillContainer/F_VN_FillContainer_TcVnPoint2_LREAL

	{attribute 'TcIecLibraryType'}
	{attribute 'external_name' := 'F_VN_FillContainer_TcVnPoint2_LREAL_GUID_29B7534F_2609_BE1D_7374_7E3A394A4CDC'}
	(* Fill the container with the specified value. Only possible for containers with basic elements. *)
	FUNCTION F_VN_FillContainer_TcVnPoint2_LREAL : HRESULT
	VAR_INPUT
		ipContainer	:	ITcVnContainer;	(* Container with basic elements *)
	END_VAR
	VAR_IN_OUT
		aValue	:	TcVnPoint2_LREAL;	(* Value to set the container elements *)
	END_VAR
	VAR_INPUT
		hrPrev	:	HRESULT;	(* HRESULT indicating the result of previous operations (If SUCCEEDED(hrPrev) equals false, no operation is executed.) *)
	END_VAR

END_FUNCTION

// Functions/Basic Container Operations/F_VN_FillContainer/F_VN_FillContainer_TcVnPoint2_REAL

	{attribute 'TcIecLibraryType'}
	{attribute 'external_name' := 'F_VN_FillContainer_TcVnPoint2_REAL_GUID_8606EFE5_F83E_B4DF_5C90_15B97636ABEF'}
	(* Fill the container with the specified value. Only possible for containers with basic elements. *)
	FUNCTION F_VN_FillContainer_TcVnPoint2_REAL : HRESULT
	VAR_INPUT
		ipContainer	:	ITcVnContainer;	(* Container with basic elements *)
	END_VAR
	VAR_IN_OUT
		aValue	:	TcVnPoint2_REAL;	(* Value to set the container elements *)
	END_VAR
	VAR_INPUT
		hrPrev	:	HRESULT;	(* HRESULT indicating the result of previous operations (If SUCCEEDED(hrPrev) equals false, no operation is executed.) *)
	END_VAR

END_FUNCTION

// Functions/Basic Container Operations/F_VN_FillContainer/F_VN_FillContainer_TcVnPoint3_LREAL

	{attribute 'TcIecLibraryType'}
	{attribute 'external_name' := 'F_VN_FillContainer_TcVnPoint3_LREAL_GUID_7D46AA72_FF7B_B0AA_6A43_30D8D3D36C59'}
	(* Fill the container with the specified value. Only possible for containers with basic elements. *)
	FUNCTION F_VN_FillContainer_TcVnPoint3_LREAL : HRESULT
	VAR_INPUT
		ipContainer	:	ITcVnContainer;	(* Container with basic elements *)
	END_VAR
	VAR_IN_OUT
		aValue	:	TcVnPoint3_LREAL;	(* Value to set the container elements *)
	END_VAR
	VAR_INPUT
		hrPrev	:	HRESULT;	(* HRESULT indicating the result of previous operations (If SUCCEEDED(hrPrev) equals false, no operation is executed.) *)
	END_VAR

END_FUNCTION

// Functions/Basic Container Operations/F_VN_FillContainer/F_VN_FillContainer_TcVnPoint3_REAL

	{attribute 'TcIecLibraryType'}
	{attribute 'external_name' := 'F_VN_FillContainer_TcVnPoint3_REAL_GUID_9CCF4901_90C4_B110_50ED_29FE74A0E11A'}
	(* Fill the container with the specified value. Only possible for containers with basic elements. *)
	FUNCTION F_VN_FillContainer_TcVnPoint3_REAL : HRESULT
	VAR_INPUT
		ipContainer	:	ITcVnContainer;	(* Container with basic elements *)
	END_VAR
	VAR_IN_OUT
		aValue	:	TcVnPoint3_REAL;	(* Value to set the container elements *)
	END_VAR
	VAR_INPUT
		hrPrev	:	HRESULT;	(* HRESULT indicating the result of previous operations (If SUCCEEDED(hrPrev) equals false, no operation is executed.) *)
	END_VAR

END_FUNCTION

// Functions/Basic Container Operations/F_VN_FillContainer/F_VN_FillContainer_TcVnRectangle_DINT

	{attribute 'TcIecLibraryType'}
	{attribute 'external_name' := 'F_VN_FillContainer_TcVnRectangle_DINT_GUID_EC066AED_D9B3_BDE1_74F2_0ED1A65DA7FC'}
	(* Fill the container with the specified value. Only possible for containers with basic elements. *)
	FUNCTION F_VN_FillContainer_TcVnRectangle_DINT : HRESULT
	VAR_INPUT
		ipContainer	:	ITcVnContainer;	(* Container with basic elements *)
	END_VAR
	VAR_IN_OUT
		stValue	:	TcVnRectangle_DINT;	(* Value to set the container elements *)
	END_VAR
	VAR_INPUT
		hrPrev	:	HRESULT;	(* HRESULT indicating the result of previous operations (If SUCCEEDED(hrPrev) equals false, no operation is executed.) *)
	END_VAR

END_FUNCTION

// Functions/Basic Container Operations/F_VN_FillContainer/F_VN_FillContainer_TcVnVector2_DINT

	{attribute 'TcIecLibraryType'}
	{attribute 'external_name' := 'F_VN_FillContainer_TcVnVector2_DINT_GUID_D692635E_7568_B79B_73CA_6A9CB31C3B47'}
	(* Fill the container with the specified value. Only possible for containers with basic elements. *)
	FUNCTION F_VN_FillContainer_TcVnVector2_DINT : HRESULT
	VAR_INPUT
		ipContainer	:	ITcVnContainer;	(* Container with basic elements *)
	END_VAR
	VAR_IN_OUT
		aValue	:	TcVnVector2_DINT;	(* Value to set the container elements *)
	END_VAR
	VAR_INPUT
		hrPrev	:	HRESULT;	(* HRESULT indicating the result of previous operations (If SUCCEEDED(hrPrev) equals false, no operation is executed.) *)
	END_VAR

END_FUNCTION

// Functions/Basic Container Operations/F_VN_FillContainer/F_VN_FillContainer_TcVnVector2_INT

	{attribute 'TcIecLibraryType'}
	{attribute 'external_name' := 'F_VN_FillContainer_TcVnVector2_INT_GUID_063210D3_CD39_BA2F_45DD_7A2D511717B9'}
	(* Fill the container with the specified value. Only possible for containers with basic elements. *)
	FUNCTION F_VN_FillContainer_TcVnVector2_INT : HRESULT
	VAR_INPUT
		ipContainer	:	ITcVnContainer;	(* Container with basic elements *)
	END_VAR
	VAR_IN_OUT
		aValue	:	TcVnVector2_INT;	(* Value to set the container elements *)
	END_VAR
	VAR_INPUT
		hrPrev	:	HRESULT;	(* HRESULT indicating the result of previous operations (If SUCCEEDED(hrPrev) equals false, no operation is executed.) *)
	END_VAR

END_FUNCTION

// Functions/Basic Container Operations/F_VN_FillContainer/F_VN_FillContainer_TcVnVector2_REAL

	{attribute 'TcIecLibraryType'}
	{attribute 'external_name' := 'F_VN_FillContainer_TcVnVector2_REAL_GUID_4153044C_6B26_B924_40C0_95C4BC703123'}
	(* Fill the container with the specified value. Only possible for containers with basic elements. *)
	FUNCTION F_VN_FillContainer_TcVnVector2_REAL : HRESULT
	VAR_INPUT
		ipContainer	:	ITcVnContainer;	(* Container with basic elements *)
	END_VAR
	VAR_IN_OUT
		aValue	:	TcVnVector2_REAL;	(* Value to set the container elements *)
	END_VAR
	VAR_INPUT
		hrPrev	:	HRESULT;	(* HRESULT indicating the result of previous operations (If SUCCEEDED(hrPrev) equals false, no operation is executed.) *)
	END_VAR

END_FUNCTION

// Functions/Basic Container Operations/F_VN_FillContainer/F_VN_FillContainer_TcVnVector2_SINT

	{attribute 'TcIecLibraryType'}
	{attribute 'external_name' := 'F_VN_FillContainer_TcVnVector2_SINT_GUID_F6D2A5D8_8722_B611_544B_6387201831CB'}
	(* Fill the container with the specified value. Only possible for containers with basic elements. *)
	FUNCTION F_VN_FillContainer_TcVnVector2_SINT : HRESULT
	VAR_INPUT
		ipContainer	:	ITcVnContainer;	(* Container with basic elements *)
	END_VAR
	VAR_IN_OUT
		aValue	:	TcVnVector2_SINT;	(* Value to set the container elements *)
	END_VAR
	VAR_INPUT
		hrPrev	:	HRESULT;	(* HRESULT indicating the result of previous operations (If SUCCEEDED(hrPrev) equals false, no operation is executed.) *)
	END_VAR

END_FUNCTION

// Functions/Basic Container Operations/F_VN_FillContainer/F_VN_FillContainer_TcVnVector2_UINT

	{attribute 'TcIecLibraryType'}
	{attribute 'external_name' := 'F_VN_FillContainer_TcVnVector2_UINT_GUID_76CC610C_CACE_BDE7_6E93_E454D8FBF2F6'}
	(* Fill the container with the specified value. Only possible for containers with basic elements. *)
	FUNCTION F_VN_FillContainer_TcVnVector2_UINT : HRESULT
	VAR_INPUT
		ipContainer	:	ITcVnContainer;	(* Container with basic elements *)
	END_VAR
	VAR_IN_OUT
		aValue	:	TcVnVector2_UINT;	(* Value to set the container elements *)
	END_VAR
	VAR_INPUT
		hrPrev	:	HRESULT;	(* HRESULT indicating the result of previous operations (If SUCCEEDED(hrPrev) equals false, no operation is executed.) *)
	END_VAR

END_FUNCTION

// Functions/Basic Container Operations/F_VN_FillContainer/F_VN_FillContainer_TcVnVector2_USINT

	{attribute 'TcIecLibraryType'}
	{attribute 'external_name' := 'F_VN_FillContainer_TcVnVector2_USINT_GUID_5E0CAADB_5624_B34E_682F_2C79CB6EAC06'}
	(* Fill the container with the specified value. Only possible for containers with basic elements. *)
	FUNCTION F_VN_FillContainer_TcVnVector2_USINT : HRESULT
	VAR_INPUT
		ipContainer	:	ITcVnContainer;	(* Container with basic elements *)
	END_VAR
	VAR_IN_OUT
		aValue	:	TcVnVector2_USINT;	(* Value to set the container elements *)
	END_VAR
	VAR_INPUT
		hrPrev	:	HRESULT;	(* HRESULT indicating the result of previous operations (If SUCCEEDED(hrPrev) equals false, no operation is executed.) *)
	END_VAR

END_FUNCTION

// Functions/Basic Container Operations/F_VN_FillContainer/F_VN_FillContainer_TcVnVector3_INT

	{attribute 'TcIecLibraryType'}
	{attribute 'external_name' := 'F_VN_FillContainer_TcVnVector3_INT_GUID_9DCC1202_147C_B357_4602_2E85C80B5341'}
	(* Fill the container with the specified value. Only possible for containers with basic elements. *)
	FUNCTION F_VN_FillContainer_TcVnVector3_INT : HRESULT
	VAR_INPUT
		ipContainer	:	ITcVnContainer;	(* Container with basic elements *)
	END_VAR
	VAR_IN_OUT
		aValue	:	TcVnVector3_INT;	(* Value to set the container elements *)
	END_VAR
	VAR_INPUT
		hrPrev	:	HRESULT;	(* HRESULT indicating the result of previous operations (If SUCCEEDED(hrPrev) equals false, no operation is executed.) *)
	END_VAR

END_FUNCTION

// Functions/Basic Container Operations/F_VN_FillContainer/F_VN_FillContainer_TcVnVector3_REAL

	{attribute 'TcIecLibraryType'}
	{attribute 'external_name' := 'F_VN_FillContainer_TcVnVector3_REAL_GUID_18B54118_1FFA_B0D2_7E39_381571834A95'}
	(* Fill the container with the specified value. Only possible for containers with basic elements. *)
	FUNCTION F_VN_FillContainer_TcVnVector3_REAL : HRESULT
	VAR_INPUT
		ipContainer	:	ITcVnContainer;	(* Container with basic elements *)
	END_VAR
	VAR_IN_OUT
		aValue	:	TcVnVector3_REAL;	(* Value to set the container elements *)
	END_VAR
	VAR_INPUT
		hrPrev	:	HRESULT;	(* HRESULT indicating the result of previous operations (If SUCCEEDED(hrPrev) equals false, no operation is executed.) *)
	END_VAR

END_FUNCTION

// Functions/Basic Container Operations/F_VN_FillContainer/F_VN_FillContainer_TcVnVector3_SINT

	{attribute 'TcIecLibraryType'}
	{attribute 'external_name' := 'F_VN_FillContainer_TcVnVector3_SINT_GUID_F18DA301_C698_BBB0_64D3_0F87AEB3FE5B'}
	(* Fill the container with the specified value. Only possible for containers with basic elements. *)
	FUNCTION F_VN_FillContainer_TcVnVector3_SINT : HRESULT
	VAR_INPUT
		ipContainer	:	ITcVnContainer;	(* Container with basic elements *)
	END_VAR
	VAR_IN_OUT
		aValue	:	TcVnVector3_SINT;	(* Value to set the container elements *)
	END_VAR
	VAR_INPUT
		hrPrev	:	HRESULT;	(* HRESULT indicating the result of previous operations (If SUCCEEDED(hrPrev) equals false, no operation is executed.) *)
	END_VAR

END_FUNCTION

// Functions/Basic Container Operations/F_VN_FillContainer/F_VN_FillContainer_TcVnVector3_UINT

	{attribute 'TcIecLibraryType'}
	{attribute 'external_name' := 'F_VN_FillContainer_TcVnVector3_UINT_GUID_C8E2BAAD_F331_BF8B_5FB9_86ED84CA7799'}
	(* Fill the container with the specified value. Only possible for containers with basic elements. *)
	FUNCTION F_VN_FillContainer_TcVnVector3_UINT : HRESULT
	VAR_INPUT
		ipContainer	:	ITcVnContainer;	(* Container with basic elements *)
	END_VAR
	VAR_IN_OUT
		aValue	:	TcVnVector3_UINT;	(* Value to set the container elements *)
	END_VAR
	VAR_INPUT
		hrPrev	:	HRESULT;	(* HRESULT indicating the result of previous operations (If SUCCEEDED(hrPrev) equals false, no operation is executed.) *)
	END_VAR

END_FUNCTION

// Functions/Basic Container Operations/F_VN_FillContainer/F_VN_FillContainer_TcVnVector3_USINT

	{attribute 'TcIecLibraryType'}
	{attribute 'external_name' := 'F_VN_FillContainer_TcVnVector3_USINT_GUID_AF7CFDA9_CF1C_BDFD_6640_B782D5C65954'}
	(* Fill the container with the specified value. Only possible for containers with basic elements. *)
	FUNCTION F_VN_FillContainer_TcVnVector3_USINT : HRESULT
	VAR_INPUT
		ipContainer	:	ITcVnContainer;	(* Container with basic elements *)
	END_VAR
	VAR_IN_OUT
		aValue	:	TcVnVector3_USINT;	(* Value to set the container elements *)
	END_VAR
	VAR_INPUT
		hrPrev	:	HRESULT;	(* HRESULT indicating the result of previous operations (If SUCCEEDED(hrPrev) equals false, no operation is executed.) *)
	END_VAR

END_FUNCTION

// Functions/Basic Container Operations/F_VN_FillContainer/F_VN_FillContainer_TcVnVector4_DINT

	{attribute 'TcIecLibraryType'}
	{attribute 'external_name' := 'F_VN_FillContainer_TcVnVector4_DINT_GUID_1794D43B_A22F_B7F2_586B_0A6ECCF48A7A'}
	(* Fill the container with the specified value. Only possible for containers with basic elements. *)
	FUNCTION F_VN_FillContainer_TcVnVector4_DINT : HRESULT
	VAR_INPUT
		ipContainer	:	ITcVnContainer;	(* Container with basic elements *)
	END_VAR
	VAR_IN_OUT
		aValue	:	TcVnVector4_DINT;	(* Value to set the container elements *)
	END_VAR
	VAR_INPUT
		hrPrev	:	HRESULT;	(* HRESULT indicating the result of previous operations (If SUCCEEDED(hrPrev) equals false, no operation is executed.) *)
	END_VAR

END_FUNCTION

// Functions/Basic Container Operations/F_VN_FillContainer/F_VN_FillContainer_TcVnVector4_INT

	{attribute 'TcIecLibraryType'}
	{attribute 'external_name' := 'F_VN_FillContainer_TcVnVector4_INT_GUID_C9254B62_51B3_B01A_4959_31F3E6B1EBF9'}
	(* Fill the container with the specified value. Only possible for containers with basic elements. *)
	FUNCTION F_VN_FillContainer_TcVnVector4_INT : HRESULT
	VAR_INPUT
		ipContainer	:	ITcVnContainer;	(* Container with basic elements *)
	END_VAR
	VAR_IN_OUT
		aValue	:	TcVnVector4_INT;	(* Value to set the container elements *)
	END_VAR
	VAR_INPUT
		hrPrev	:	HRESULT;	(* HRESULT indicating the result of previous operations (If SUCCEEDED(hrPrev) equals false, no operation is executed.) *)
	END_VAR

END_FUNCTION

// Functions/Basic Container Operations/F_VN_FillContainer/F_VN_FillContainer_TcVnVector4_LREAL

	{attribute 'TcIecLibraryType'}
	{attribute 'external_name' := 'F_VN_FillContainer_TcVnVector4_LREAL_GUID_CE144EC9_0740_BEC9_6BA6_50B049DD7E1E'}
	(* Fill the container with the specified value. Only possible for containers with basic elements. *)
	FUNCTION F_VN_FillContainer_TcVnVector4_LREAL : HRESULT
	VAR_INPUT
		ipContainer	:	ITcVnContainer;	(* Container with basic elements *)
	END_VAR
	VAR_IN_OUT
		aValue	:	TcVnVector4_LREAL;	(* Value to set the container elements *)
	END_VAR
	VAR_INPUT
		hrPrev	:	HRESULT;	(* HRESULT indicating the result of previous operations (If SUCCEEDED(hrPrev) equals false, no operation is executed.) *)
	END_VAR

END_FUNCTION

// Functions/Basic Container Operations/F_VN_FillContainer/F_VN_FillContainer_TcVnVector4_SINT

	{attribute 'TcIecLibraryType'}
	{attribute 'external_name' := 'F_VN_FillContainer_TcVnVector4_SINT_GUID_3DE67987_9DEF_B3B5_4EF6_060BE849E3C9'}
	(* Fill the container with the specified value. Only possible for containers with basic elements. *)
	FUNCTION F_VN_FillContainer_TcVnVector4_SINT : HRESULT
	VAR_INPUT
		ipContainer	:	ITcVnContainer;	(* Container with basic elements *)
	END_VAR
	VAR_IN_OUT
		aValue	:	TcVnVector4_SINT;	(* Value to set the container elements *)
	END_VAR
	VAR_INPUT
		hrPrev	:	HRESULT;	(* HRESULT indicating the result of previous operations (If SUCCEEDED(hrPrev) equals false, no operation is executed.) *)
	END_VAR

END_FUNCTION

// Functions/Basic Container Operations/F_VN_FillContainer/F_VN_FillContainer_TcVnVector4_UINT

	{attribute 'TcIecLibraryType'}
	{attribute 'external_name' := 'F_VN_FillContainer_TcVnVector4_UINT_GUID_F0D6F306_12AD_B70F_7850_C05E73A00382'}
	(* Fill the container with the specified value. Only possible for containers with basic elements. *)
	FUNCTION F_VN_FillContainer_TcVnVector4_UINT : HRESULT
	VAR_INPUT
		ipContainer	:	ITcVnContainer;	(* Container with basic elements *)
	END_VAR
	VAR_IN_OUT
		aValue	:	TcVnVector4_UINT;	(* Value to set the container elements *)
	END_VAR
	VAR_INPUT
		hrPrev	:	HRESULT;	(* HRESULT indicating the result of previous operations (If SUCCEEDED(hrPrev) equals false, no operation is executed.) *)
	END_VAR

END_FUNCTION

// Functions/Basic Container Operations/F_VN_FillContainer/F_VN_FillContainer_TcVnVector4_USINT

	{attribute 'TcIecLibraryType'}
	{attribute 'external_name' := 'F_VN_FillContainer_TcVnVector4_USINT_GUID_2128C026_89CA_B364_530F_32EEAB00E1DE'}
	(* Fill the container with the specified value. Only possible for containers with basic elements. *)
	FUNCTION F_VN_FillContainer_TcVnVector4_USINT : HRESULT
	VAR_INPUT
		ipContainer	:	ITcVnContainer;	(* Container with basic elements *)
	END_VAR
	VAR_IN_OUT
		aValue	:	TcVnVector4_USINT;	(* Value to set the container elements *)
	END_VAR
	VAR_INPUT
		hrPrev	:	HRESULT;	(* HRESULT indicating the result of previous operations (If SUCCEEDED(hrPrev) equals false, no operation is executed.) *)
	END_VAR

END_FUNCTION

// Functions/Basic Container Operations/F_VN_FillContainer/F_VN_FillContainer_UDINT

	{attribute 'TcIecLibraryType'}
	{attribute 'external_name' := 'F_VN_FillContainer_UDINT_GUID_A01B9964_AE80_B769_728B_A109218542BF'}
	(* Fill the container with the specified value. Only possible for containers with basic elements. *)
	FUNCTION F_VN_FillContainer_UDINT : HRESULT
	VAR_INPUT
		ipContainer	:	ITcVnContainer;	(* Container with basic elements *)
		nValue	:	UDINT;	(* Value to set the container elements *)
		hrPrev	:	HRESULT;	(* HRESULT indicating the result of previous operations (If SUCCEEDED(hrPrev) equals false, no operation is executed.) *)
	END_VAR

END_FUNCTION

// Functions/Basic Container Operations/F_VN_FillContainer/F_VN_FillContainer_UINT

	{attribute 'TcIecLibraryType'}
	{attribute 'external_name' := 'F_VN_FillContainer_UINT_GUID_36442DC0_CF51_B8F9_6D0A_D59281BD25BC'}
	(* Fill the container with the specified value. Only possible for containers with basic elements. *)
	FUNCTION F_VN_FillContainer_UINT : HRESULT
	VAR_INPUT
		ipContainer	:	ITcVnContainer;	(* Container with basic elements *)
		nValue	:	UINT;	(* Value to set the container elements *)
		hrPrev	:	HRESULT;	(* HRESULT indicating the result of previous operations (If SUCCEEDED(hrPrev) equals false, no operation is executed.) *)
	END_VAR

END_FUNCTION

// Functions/Basic Container Operations/F_VN_FillContainer/F_VN_FillContainer_ULINT

	{attribute 'TcIecLibraryType'}
	{attribute 'external_name' := 'F_VN_FillContainer_ULINT_GUID_9D930F59_7243_B488_561C_87D45212EEDF'}
	(* Fill the container with the specified value. Only possible for containers with basic elements. *)
	FUNCTION F_VN_FillContainer_ULINT : HRESULT
	VAR_INPUT
		ipContainer	:	ITcVnContainer;	(* Container with basic elements *)
		nValue	:	ULINT;	(* Value to set the container elements *)
		hrPrev	:	HRESULT;	(* HRESULT indicating the result of previous operations (If SUCCEEDED(hrPrev) equals false, no operation is executed.) *)
	END_VAR

END_FUNCTION

// Functions/Basic Container Operations/F_VN_FillContainer/F_VN_FillContainer_USINT

	{attribute 'TcIecLibraryType'}
	{attribute 'external_name' := 'F_VN_FillContainer_USINT_GUID_F7633142_EBFD_B1D7_5A30_FDD1946AF78D'}
	(* Fill the container with the specified value. Only possible for containers with basic elements. *)
	FUNCTION F_VN_FillContainer_USINT : HRESULT
	VAR_INPUT
		ipContainer	:	ITcVnContainer;	(* Container with basic elements *)
		nValue	:	USINT;	(* Value to set the container elements *)
		hrPrev	:	HRESULT;	(* HRESULT indicating the result of previous operations (If SUCCEEDED(hrPrev) equals false, no operation is executed.) *)
	END_VAR

END_FUNCTION

// Functions/Basic Container Operations/F_VN_FillContainerExp/F_VN_FillContainerExp_DINT

	{attribute 'TcIecLibraryType'}
	{attribute 'external_name' := 'F_VN_FillContainerExp_DINT_GUID_4CF619BF_65BE_B6F3_5941_0774F4AA65C5'}
	(* Partially fill the container with the specified value. Only possible for containers with basic elements. (expert function) *)
	FUNCTION F_VN_FillContainerExp_DINT : HRESULT
	VAR_INPUT
		ipContainer	:	ITcVnContainer;	(* Container with basic elements *)
		nValue	:	DINT;	(* Value to set the container elements *)
		nStartIdx	:	ULINT;	(* Start index *)
		nCount	:	ULINT;	(* Number of elements to set *)
		hrPrev	:	HRESULT;	(* HRESULT indicating the result of previous operations (If SUCCEEDED(hrPrev) equals false, no operation is executed.) *)
	END_VAR

END_FUNCTION

// Functions/Basic Container Operations/F_VN_FillContainerExp/F_VN_FillContainerExp_INT

	{attribute 'TcIecLibraryType'}
	{attribute 'external_name' := 'F_VN_FillContainerExp_INT_GUID_57276027_1E5E_B0E6_4419_BE69EF3D7C71'}
	(* Partially fill the container with the specified value. Only possible for containers with basic elements. (expert function) *)
	FUNCTION F_VN_FillContainerExp_INT : HRESULT
	VAR_INPUT
		ipContainer	:	ITcVnContainer;	(* Container with basic elements *)
		nValue	:	INT;	(* Value to set the container elements *)
		nStartIdx	:	ULINT;	(* Start index *)
		nCount	:	ULINT;	(* Number of elements to set *)
		hrPrev	:	HRESULT;	(* HRESULT indicating the result of previous operations (If SUCCEEDED(hrPrev) equals false, no operation is executed.) *)
	END_VAR

END_FUNCTION

// Functions/Basic Container Operations/F_VN_FillContainerExp/F_VN_FillContainerExp_ITcVnImage

	{attribute 'TcIecLibraryType'}
	{attribute 'external_name' := 'F_VN_FillContainerExp_ITcVnImage_GUID_62528B5F_44C8_B4B1_44F1_617538E60937'}
	(* Partially fill the container with the specified value. Only possible for containers with basic elements. (expert function) *)
	FUNCTION F_VN_FillContainerExp_ITcVnImage : HRESULT
	VAR_INPUT
		ipContainer	:	ITcVnContainer;	(* Container with basic elements *)
		ipValue	:	ITcVnImage;	(* Value to set the container elements *)
		nStartIdx	:	ULINT;	(* Start index *)
		nCount	:	ULINT;	(* Number of elements to set *)
		hrPrev	:	HRESULT;	(* HRESULT indicating the result of previous operations (If SUCCEEDED(hrPrev) equals false, no operation is executed.) *)
	END_VAR

END_FUNCTION

// Functions/Basic Container Operations/F_VN_FillContainerExp/F_VN_FillContainerExp_LREAL

	{attribute 'TcIecLibraryType'}
	{attribute 'external_name' := 'F_VN_FillContainerExp_LREAL_GUID_F2898D42_7A52_B81A_514F_F77B21EAD703'}
	(* Partially fill the container with the specified value. Only possible for containers with basic elements. (expert function) *)
	FUNCTION F_VN_FillContainerExp_LREAL : HRESULT
	VAR_INPUT
		ipContainer	:	ITcVnContainer;	(* Container with basic elements *)
		fValue	:	LREAL;	(* Value to set the container elements *)
		nStartIdx	:	ULINT;	(* Start index *)
		nCount	:	ULINT;	(* Number of elements to set *)
		hrPrev	:	HRESULT;	(* HRESULT indicating the result of previous operations (If SUCCEEDED(hrPrev) equals false, no operation is executed.) *)
	END_VAR

END_FUNCTION

// Functions/Basic Container Operations/F_VN_FillContainerExp/F_VN_FillContainerExp_REAL

	{attribute 'TcIecLibraryType'}
	{attribute 'external_name' := 'F_VN_FillContainerExp_REAL_GUID_BC993E55_6086_BBD0_618A_60859B6EAED0'}
	(* Partially fill the container with the specified value. Only possible for containers with basic elements. (expert function) *)
	FUNCTION F_VN_FillContainerExp_REAL : HRESULT
	VAR_INPUT
		ipContainer	:	ITcVnContainer;	(* Container with basic elements *)
		fValue	:	REAL;	(* Value to set the container elements *)
		nStartIdx	:	ULINT;	(* Start index *)
		nCount	:	ULINT;	(* Number of elements to set *)
		hrPrev	:	HRESULT;	(* HRESULT indicating the result of previous operations (If SUCCEEDED(hrPrev) equals false, no operation is executed.) *)
	END_VAR

END_FUNCTION

// Functions/Basic Container Operations/F_VN_FillContainerExp/F_VN_FillContainerExp_SINT

	{attribute 'TcIecLibraryType'}
	{attribute 'external_name' := 'F_VN_FillContainerExp_SINT_GUID_64A7445E_E7D0_B6DC_6B7E_D799AAB92AB4'}
	(* Partially fill the container with the specified value. Only possible for containers with basic elements. (expert function) *)
	FUNCTION F_VN_FillContainerExp_SINT : HRESULT
	VAR_INPUT
		ipContainer	:	ITcVnContainer;	(* Container with basic elements *)
		nValue	:	SINT;	(* Value to set the container elements *)
		nStartIdx	:	ULINT;	(* Start index *)
		nCount	:	ULINT;	(* Number of elements to set *)
		hrPrev	:	HRESULT;	(* HRESULT indicating the result of previous operations (If SUCCEEDED(hrPrev) equals false, no operation is executed.) *)
	END_VAR

END_FUNCTION

// Functions/Basic Container Operations/F_VN_FillContainerExp/F_VN_FillContainerExp_TcVnDMatch

	{attribute 'TcIecLibraryType'}
	{attribute 'external_name' := 'F_VN_FillContainerExp_TcVnDMatch_GUID_9A9251BE_6FB8_B65D_7C5B_0D2B37899506'}
	(* Partially fill the container with the specified value. Only possible for containers with basic elements. (expert function) *)
	FUNCTION F_VN_FillContainerExp_TcVnDMatch : HRESULT
	VAR_INPUT
		ipContainer	:	ITcVnContainer;	(* Container with basic elements *)
	END_VAR
	VAR_IN_OUT
		stValue	:	TcVnDMatch;	(* Value to set the container elements *)
	END_VAR
	VAR_INPUT
		nStartIdx	:	ULINT;	(* Start index *)
		nCount	:	ULINT;	(* Number of elements to set *)
		hrPrev	:	HRESULT;	(* HRESULT indicating the result of previous operations (If SUCCEEDED(hrPrev) equals false, no operation is executed.) *)
	END_VAR

END_FUNCTION

// Functions/Basic Container Operations/F_VN_FillContainerExp/F_VN_FillContainerExp_TcVnKeyPoint

	{attribute 'TcIecLibraryType'}
	{attribute 'external_name' := 'F_VN_FillContainerExp_TcVnKeyPoint_GUID_AAAD9C01_798D_BA6A_5838_6B483EF932EB'}
	(* Partially fill the container with the specified value. Only possible for containers with basic elements. (expert function) *)
	FUNCTION F_VN_FillContainerExp_TcVnKeyPoint : HRESULT
	VAR_INPUT
		ipContainer	:	ITcVnContainer;	(* Container with basic elements *)
	END_VAR
	VAR_IN_OUT
		stValue	:	TcVnKeyPoint;	(* Value to set the container elements *)
	END_VAR
	VAR_INPUT
		nStartIdx	:	ULINT;	(* Start index *)
		nCount	:	ULINT;	(* Number of elements to set *)
		hrPrev	:	HRESULT;	(* HRESULT indicating the result of previous operations (If SUCCEEDED(hrPrev) equals false, no operation is executed.) *)
	END_VAR

END_FUNCTION

// Functions/Basic Container Operations/F_VN_FillContainerExp/F_VN_FillContainerExp_TcVnPoint2_DINT

	{attribute 'TcIecLibraryType'}
	{attribute 'external_name' := 'F_VN_FillContainerExp_TcVnPoint2_DINT_GUID_A1D8FB04_419D_B618_46B2_F37C2B21420B'}
	(* Partially fill the container with the specified value. Only possible for containers with basic elements. (expert function) *)
	FUNCTION F_VN_FillContainerExp_TcVnPoint2_DINT : HRESULT
	VAR_INPUT
		ipContainer	:	ITcVnContainer;	(* Container with basic elements *)
	END_VAR
	VAR_IN_OUT
		aValue	:	TcVnPoint2_DINT;	(* Value to set the container elements *)
	END_VAR
	VAR_INPUT
		nStartIdx	:	ULINT;	(* Start index *)
		nCount	:	ULINT;	(* Number of elements to set *)
		hrPrev	:	HRESULT;	(* HRESULT indicating the result of previous operations (If SUCCEEDED(hrPrev) equals false, no operation is executed.) *)
	END_VAR

END_FUNCTION

// Functions/Basic Container Operations/F_VN_FillContainerExp/F_VN_FillContainerExp_TcVnPoint2_LREAL

	{attribute 'TcIecLibraryType'}
	{attribute 'external_name' := 'F_VN_FillContainerExp_TcVnPoint2_LREAL_GUID_1BD0C868_A64F_B0CC_7866_4200B89F1518'}
	(* Partially fill the container with the specified value. Only possible for containers with basic elements. (expert function) *)
	FUNCTION F_VN_FillContainerExp_TcVnPoint2_LREAL : HRESULT
	VAR_INPUT
		ipContainer	:	ITcVnContainer;	(* Container with basic elements *)
	END_VAR
	VAR_IN_OUT
		aValue	:	TcVnPoint2_LREAL;	(* Value to set the container elements *)
	END_VAR
	VAR_INPUT
		nStartIdx	:	ULINT;	(* Start index *)
		nCount	:	ULINT;	(* Number of elements to set *)
		hrPrev	:	HRESULT;	(* HRESULT indicating the result of previous operations (If SUCCEEDED(hrPrev) equals false, no operation is executed.) *)
	END_VAR

END_FUNCTION

// Functions/Basic Container Operations/F_VN_FillContainerExp/F_VN_FillContainerExp_TcVnPoint2_REAL

	{attribute 'TcIecLibraryType'}
	{attribute 'external_name' := 'F_VN_FillContainerExp_TcVnPoint2_REAL_GUID_26B46AE5_7C96_B539_724E_878E80DE3DE3'}
	(* Partially fill the container with the specified value. Only possible for containers with basic elements. (expert function) *)
	FUNCTION F_VN_FillContainerExp_TcVnPoint2_REAL : HRESULT
	VAR_INPUT
		ipContainer	:	ITcVnContainer;	(* Container with basic elements *)
	END_VAR
	VAR_IN_OUT
		aValue	:	TcVnPoint2_REAL;	(* Value to set the container elements *)
	END_VAR
	VAR_INPUT
		nStartIdx	:	ULINT;	(* Start index *)
		nCount	:	ULINT;	(* Number of elements to set *)
		hrPrev	:	HRESULT;	(* HRESULT indicating the result of previous operations (If SUCCEEDED(hrPrev) equals false, no operation is executed.) *)
	END_VAR

END_FUNCTION

// Functions/Basic Container Operations/F_VN_FillContainerExp/F_VN_FillContainerExp_TcVnPoint3_LREAL

	{attribute 'TcIecLibraryType'}
	{attribute 'external_name' := 'F_VN_FillContainerExp_TcVnPoint3_LREAL_GUID_4349C908_0AE5_B31D_66A9_FA40ACE02DE6'}
	(* Partially fill the container with the specified value. Only possible for containers with basic elements. (expert function) *)
	FUNCTION F_VN_FillContainerExp_TcVnPoint3_LREAL : HRESULT
	VAR_INPUT
		ipContainer	:	ITcVnContainer;	(* Container with basic elements *)
	END_VAR
	VAR_IN_OUT
		aValue	:	TcVnPoint3_LREAL;	(* Value to set the container elements *)
	END_VAR
	VAR_INPUT
		nStartIdx	:	ULINT;	(* Start index *)
		nCount	:	ULINT;	(* Number of elements to set *)
		hrPrev	:	HRESULT;	(* HRESULT indicating the result of previous operations (If SUCCEEDED(hrPrev) equals false, no operation is executed.) *)
	END_VAR

END_FUNCTION

// Functions/Basic Container Operations/F_VN_FillContainerExp/F_VN_FillContainerExp_TcVnPoint3_REAL

	{attribute 'TcIecLibraryType'}
	{attribute 'external_name' := 'F_VN_FillContainerExp_TcVnPoint3_REAL_GUID_9EF5B2E0_CB3A_B323_6F5E_D75507B68F20'}
	(* Partially fill the container with the specified value. Only possible for containers with basic elements. (expert function) *)
	FUNCTION F_VN_FillContainerExp_TcVnPoint3_REAL : HRESULT
	VAR_INPUT
		ipContainer	:	ITcVnContainer;	(* Container with basic elements *)
	END_VAR
	VAR_IN_OUT
		aValue	:	TcVnPoint3_REAL;	(* Value to set the container elements *)
	END_VAR
	VAR_INPUT
		nStartIdx	:	ULINT;	(* Start index *)
		nCount	:	ULINT;	(* Number of elements to set *)
		hrPrev	:	HRESULT;	(* HRESULT indicating the result of previous operations (If SUCCEEDED(hrPrev) equals false, no operation is executed.) *)
	END_VAR

END_FUNCTION

// Functions/Basic Container Operations/F_VN_FillContainerExp/F_VN_FillContainerExp_TcVnRectangle_DINT

	{attribute 'TcIecLibraryType'}
	{attribute 'external_name' := 'F_VN_FillContainerExp_TcVnRectangle_DINT_GUID_7F9D5309_9BE8_B531_68D4_BFDB26E7B66B'}
	(* Partially fill the container with the specified value. Only possible for containers with basic elements. (expert function) *)
	FUNCTION F_VN_FillContainerExp_TcVnRectangle_DINT : HRESULT
	VAR_INPUT
		ipContainer	:	ITcVnContainer;	(* Container with basic elements *)
	END_VAR
	VAR_IN_OUT
		stValue	:	TcVnRectangle_DINT;	(* Value to set the container elements *)
	END_VAR
	VAR_INPUT
		nStartIdx	:	ULINT;	(* Start index *)
		nCount	:	ULINT;	(* Number of elements to set *)
		hrPrev	:	HRESULT;	(* HRESULT indicating the result of previous operations (If SUCCEEDED(hrPrev) equals false, no operation is executed.) *)
	END_VAR

END_FUNCTION

// Functions/Basic Container Operations/F_VN_FillContainerExp/F_VN_FillContainerExp_TcVnVector2_DINT

	{attribute 'TcIecLibraryType'}
	{attribute 'external_name' := 'F_VN_FillContainerExp_TcVnVector2_DINT_GUID_210F13E2_2177_B782_7D70_1EF3BA6BEF12'}
	(* Partially fill the container with the specified value. Only possible for containers with basic elements. (expert function) *)
	FUNCTION F_VN_FillContainerExp_TcVnVector2_DINT : HRESULT
	VAR_INPUT
		ipContainer	:	ITcVnContainer;	(* Container with basic elements *)
	END_VAR
	VAR_IN_OUT
		aValue	:	TcVnVector2_DINT;	(* Value to set the container elements *)
	END_VAR
	VAR_INPUT
		nStartIdx	:	ULINT;	(* Start index *)
		nCount	:	ULINT;	(* Number of elements to set *)
		hrPrev	:	HRESULT;	(* HRESULT indicating the result of previous operations (If SUCCEEDED(hrPrev) equals false, no operation is executed.) *)
	END_VAR

END_FUNCTION

// Functions/Basic Container Operations/F_VN_FillContainerExp/F_VN_FillContainerExp_TcVnVector2_INT

	{attribute 'TcIecLibraryType'}
	{attribute 'external_name' := 'F_VN_FillContainerExp_TcVnVector2_INT_GUID_048A080C_010D_BEBA_4A97_C0BA1E55458C'}
	(* Partially fill the container with the specified value. Only possible for containers with basic elements. (expert function) *)
	FUNCTION F_VN_FillContainerExp_TcVnVector2_INT : HRESULT
	VAR_INPUT
		ipContainer	:	ITcVnContainer;	(* Container with basic elements *)
	END_VAR
	VAR_IN_OUT
		aValue	:	TcVnVector2_INT;	(* Value to set the container elements *)
	END_VAR
	VAR_INPUT
		nStartIdx	:	ULINT;	(* Start index *)
		nCount	:	ULINT;	(* Number of elements to set *)
		hrPrev	:	HRESULT;	(* HRESULT indicating the result of previous operations (If SUCCEEDED(hrPrev) equals false, no operation is executed.) *)
	END_VAR

END_FUNCTION

// Functions/Basic Container Operations/F_VN_FillContainerExp/F_VN_FillContainerExp_TcVnVector2_REAL

	{attribute 'TcIecLibraryType'}
	{attribute 'external_name' := 'F_VN_FillContainerExp_TcVnVector2_REAL_GUID_8DF29405_268E_B772_4A8F_32EC9F16033E'}
	(* Partially fill the container with the specified value. Only possible for containers with basic elements. (expert function) *)
	FUNCTION F_VN_FillContainerExp_TcVnVector2_REAL : HRESULT
	VAR_INPUT
		ipContainer	:	ITcVnContainer;	(* Container with basic elements *)
	END_VAR
	VAR_IN_OUT
		aValue	:	TcVnVector2_REAL;	(* Value to set the container elements *)
	END_VAR
	VAR_INPUT
		nStartIdx	:	ULINT;	(* Start index *)
		nCount	:	ULINT;	(* Number of elements to set *)
		hrPrev	:	HRESULT;	(* HRESULT indicating the result of previous operations (If SUCCEEDED(hrPrev) equals false, no operation is executed.) *)
	END_VAR

END_FUNCTION

// Functions/Basic Container Operations/F_VN_FillContainerExp/F_VN_FillContainerExp_TcVnVector2_SINT

	{attribute 'TcIecLibraryType'}
	{attribute 'external_name' := 'F_VN_FillContainerExp_TcVnVector2_SINT_GUID_AE4116C1_0E19_B28C_6DDD_FD7E52356742'}
	(* Partially fill the container with the specified value. Only possible for containers with basic elements. (expert function) *)
	FUNCTION F_VN_FillContainerExp_TcVnVector2_SINT : HRESULT
	VAR_INPUT
		ipContainer	:	ITcVnContainer;	(* Container with basic elements *)
	END_VAR
	VAR_IN_OUT
		aValue	:	TcVnVector2_SINT;	(* Value to set the container elements *)
	END_VAR
	VAR_INPUT
		nStartIdx	:	ULINT;	(* Start index *)
		nCount	:	ULINT;	(* Number of elements to set *)
		hrPrev	:	HRESULT;	(* HRESULT indicating the result of previous operations (If SUCCEEDED(hrPrev) equals false, no operation is executed.) *)
	END_VAR

END_FUNCTION

// Functions/Basic Container Operations/F_VN_FillContainerExp/F_VN_FillContainerExp_TcVnVector2_UINT

	{attribute 'TcIecLibraryType'}
	{attribute 'external_name' := 'F_VN_FillContainerExp_TcVnVector2_UINT_GUID_DCF698AB_767C_B767_5E42_5F4297A2ED82'}
	(* Partially fill the container with the specified value. Only possible for containers with basic elements. (expert function) *)
	FUNCTION F_VN_FillContainerExp_TcVnVector2_UINT : HRESULT
	VAR_INPUT
		ipContainer	:	ITcVnContainer;	(* Container with basic elements *)
	END_VAR
	VAR_IN_OUT
		aValue	:	TcVnVector2_UINT;	(* Value to set the container elements *)
	END_VAR
	VAR_INPUT
		nStartIdx	:	ULINT;	(* Start index *)
		nCount	:	ULINT;	(* Number of elements to set *)
		hrPrev	:	HRESULT;	(* HRESULT indicating the result of previous operations (If SUCCEEDED(hrPrev) equals false, no operation is executed.) *)
	END_VAR

END_FUNCTION

// Functions/Basic Container Operations/F_VN_FillContainerExp/F_VN_FillContainerExp_TcVnVector2_USINT

	{attribute 'TcIecLibraryType'}
	{attribute 'external_name' := 'F_VN_FillContainerExp_TcVnVector2_USINT_GUID_3EFF349F_1D7E_B0BF_4050_65E44C94BB7A'}
	(* Partially fill the container with the specified value. Only possible for containers with basic elements. (expert function) *)
	FUNCTION F_VN_FillContainerExp_TcVnVector2_USINT : HRESULT
	VAR_INPUT
		ipContainer	:	ITcVnContainer;	(* Container with basic elements *)
	END_VAR
	VAR_IN_OUT
		aValue	:	TcVnVector2_USINT;	(* Value to set the container elements *)
	END_VAR
	VAR_INPUT
		nStartIdx	:	ULINT;	(* Start index *)
		nCount	:	ULINT;	(* Number of elements to set *)
		hrPrev	:	HRESULT;	(* HRESULT indicating the result of previous operations (If SUCCEEDED(hrPrev) equals false, no operation is executed.) *)
	END_VAR

END_FUNCTION

// Functions/Basic Container Operations/F_VN_FillContainerExp/F_VN_FillContainerExp_TcVnVector3_INT

	{attribute 'TcIecLibraryType'}
	{attribute 'external_name' := 'F_VN_FillContainerExp_TcVnVector3_INT_GUID_7C53105C_746B_B764_60F0_EB8A3ACC083F'}
	(* Partially fill the container with the specified value. Only possible for containers with basic elements. (expert function) *)
	FUNCTION F_VN_FillContainerExp_TcVnVector3_INT : HRESULT
	VAR_INPUT
		ipContainer	:	ITcVnContainer;	(* Container with basic elements *)
	END_VAR
	VAR_IN_OUT
		aValue	:	TcVnVector3_INT;	(* Value to set the container elements *)
	END_VAR
	VAR_INPUT
		nStartIdx	:	ULINT;	(* Start index *)
		nCount	:	ULINT;	(* Number of elements to set *)
		hrPrev	:	HRESULT;	(* HRESULT indicating the result of previous operations (If SUCCEEDED(hrPrev) equals false, no operation is executed.) *)
	END_VAR

END_FUNCTION

// Functions/Basic Container Operations/F_VN_FillContainerExp/F_VN_FillContainerExp_TcVnVector3_REAL

	{attribute 'TcIecLibraryType'}
	{attribute 'external_name' := 'F_VN_FillContainerExp_TcVnVector3_REAL_GUID_033F7082_A01D_B934_4E78_5CE4549FC26A'}
	(* Partially fill the container with the specified value. Only possible for containers with basic elements. (expert function) *)
	FUNCTION F_VN_FillContainerExp_TcVnVector3_REAL : HRESULT
	VAR_INPUT
		ipContainer	:	ITcVnContainer;	(* Container with basic elements *)
	END_VAR
	VAR_IN_OUT
		aValue	:	TcVnVector3_REAL;	(* Value to set the container elements *)
	END_VAR
	VAR_INPUT
		nStartIdx	:	ULINT;	(* Start index *)
		nCount	:	ULINT;	(* Number of elements to set *)
		hrPrev	:	HRESULT;	(* HRESULT indicating the result of previous operations (If SUCCEEDED(hrPrev) equals false, no operation is executed.) *)
	END_VAR

END_FUNCTION

// Functions/Basic Container Operations/F_VN_FillContainerExp/F_VN_FillContainerExp_TcVnVector3_SINT

	{attribute 'TcIecLibraryType'}
	{attribute 'external_name' := 'F_VN_FillContainerExp_TcVnVector3_SINT_GUID_3346C628_7EE4_B5A3_5962_E448ED84600C'}
	(* Partially fill the container with the specified value. Only possible for containers with basic elements. (expert function) *)
	FUNCTION F_VN_FillContainerExp_TcVnVector3_SINT : HRESULT
	VAR_INPUT
		ipContainer	:	ITcVnContainer;	(* Container with basic elements *)
	END_VAR
	VAR_IN_OUT
		aValue	:	TcVnVector3_SINT;	(* Value to set the container elements *)
	END_VAR
	VAR_INPUT
		nStartIdx	:	ULINT;	(* Start index *)
		nCount	:	ULINT;	(* Number of elements to set *)
		hrPrev	:	HRESULT;	(* HRESULT indicating the result of previous operations (If SUCCEEDED(hrPrev) equals false, no operation is executed.) *)
	END_VAR

END_FUNCTION

// Functions/Basic Container Operations/F_VN_FillContainerExp/F_VN_FillContainerExp_TcVnVector3_UINT

	{attribute 'TcIecLibraryType'}
	{attribute 'external_name' := 'F_VN_FillContainerExp_TcVnVector3_UINT_GUID_5613BC10_C230_B86C_56FD_DF077FB05BDD'}
	(* Partially fill the container with the specified value. Only possible for containers with basic elements. (expert function) *)
	FUNCTION F_VN_FillContainerExp_TcVnVector3_UINT : HRESULT
	VAR_INPUT
		ipContainer	:	ITcVnContainer;	(* Container with basic elements *)
	END_VAR
	VAR_IN_OUT
		aValue	:	TcVnVector3_UINT;	(* Value to set the container elements *)
	END_VAR
	VAR_INPUT
		nStartIdx	:	ULINT;	(* Start index *)
		nCount	:	ULINT;	(* Number of elements to set *)
		hrPrev	:	HRESULT;	(* HRESULT indicating the result of previous operations (If SUCCEEDED(hrPrev) equals false, no operation is executed.) *)
	END_VAR

END_FUNCTION

// Functions/Basic Container Operations/F_VN_FillContainerExp/F_VN_FillContainerExp_TcVnVector3_USINT

	{attribute 'TcIecLibraryType'}
	{attribute 'external_name' := 'F_VN_FillContainerExp_TcVnVector3_USINT_GUID_5B569AB2_9918_B2AF_7F44_05638AF996E2'}
	(* Partially fill the container with the specified value. Only possible for containers with basic elements. (expert function) *)
	FUNCTION F_VN_FillContainerExp_TcVnVector3_USINT : HRESULT
	VAR_INPUT
		ipContainer	:	ITcVnContainer;	(* Container with basic elements *)
	END_VAR
	VAR_IN_OUT
		aValue	:	TcVnVector3_USINT;	(* Value to set the container elements *)
	END_VAR
	VAR_INPUT
		nStartIdx	:	ULINT;	(* Start index *)
		nCount	:	ULINT;	(* Number of elements to set *)
		hrPrev	:	HRESULT;	(* HRESULT indicating the result of previous operations (If SUCCEEDED(hrPrev) equals false, no operation is executed.) *)
	END_VAR

END_FUNCTION

// Functions/Basic Container Operations/F_VN_FillContainerExp/F_VN_FillContainerExp_TcVnVector4_DINT

	{attribute 'TcIecLibraryType'}
	{attribute 'external_name' := 'F_VN_FillContainerExp_TcVnVector4_DINT_GUID_249508C9_2F9C_B244_4306_E34DD84B261B'}
	(* Partially fill the container with the specified value. Only possible for containers with basic elements. (expert function) *)
	FUNCTION F_VN_FillContainerExp_TcVnVector4_DINT : HRESULT
	VAR_INPUT
		ipContainer	:	ITcVnContainer;	(* Container with basic elements *)
	END_VAR
	VAR_IN_OUT
		aValue	:	TcVnVector4_DINT;	(* Value to set the container elements *)
	END_VAR
	VAR_INPUT
		nStartIdx	:	ULINT;	(* Start index *)
		nCount	:	ULINT;	(* Number of elements to set *)
		hrPrev	:	HRESULT;	(* HRESULT indicating the result of previous operations (If SUCCEEDED(hrPrev) equals false, no operation is executed.) *)
	END_VAR

END_FUNCTION

// Functions/Basic Container Operations/F_VN_FillContainerExp/F_VN_FillContainerExp_TcVnVector4_INT

	{attribute 'TcIecLibraryType'}
	{attribute 'external_name' := 'F_VN_FillContainerExp_TcVnVector4_INT_GUID_0A26AD84_D484_B56B_682E_2883C89A4976'}
	(* Partially fill the container with the specified value. Only possible for containers with basic elements. (expert function) *)
	FUNCTION F_VN_FillContainerExp_TcVnVector4_INT : HRESULT
	VAR_INPUT
		ipContainer	:	ITcVnContainer;	(* Container with basic elements *)
	END_VAR
	VAR_IN_OUT
		aValue	:	TcVnVector4_INT;	(* Value to set the container elements *)
	END_VAR
	VAR_INPUT
		nStartIdx	:	ULINT;	(* Start index *)
		nCount	:	ULINT;	(* Number of elements to set *)
		hrPrev	:	HRESULT;	(* HRESULT indicating the result of previous operations (If SUCCEEDED(hrPrev) equals false, no operation is executed.) *)
	END_VAR

END_FUNCTION

// Functions/Basic Container Operations/F_VN_FillContainerExp/F_VN_FillContainerExp_TcVnVector4_LREAL

	{attribute 'TcIecLibraryType'}
	{attribute 'external_name' := 'F_VN_FillContainerExp_TcVnVector4_LREAL_GUID_2AB0095E_177A_BAB8_53C7_0AF75CEF13C9'}
	(* Partially fill the container with the specified value. Only possible for containers with basic elements. (expert function) *)
	FUNCTION F_VN_FillContainerExp_TcVnVector4_LREAL : HRESULT
	VAR_INPUT
		ipContainer	:	ITcVnContainer;	(* Container with basic elements *)
	END_VAR
	VAR_IN_OUT
		aValue	:	TcVnVector4_LREAL;	(* Value to set the container elements *)
	END_VAR
	VAR_INPUT
		nStartIdx	:	ULINT;	(* Start index *)
		nCount	:	ULINT;	(* Number of elements to set *)
		hrPrev	:	HRESULT;	(* HRESULT indicating the result of previous operations (If SUCCEEDED(hrPrev) equals false, no operation is executed.) *)
	END_VAR

END_FUNCTION

// Functions/Basic Container Operations/F_VN_FillContainerExp/F_VN_FillContainerExp_TcVnVector4_SINT

	{attribute 'TcIecLibraryType'}
	{attribute 'external_name' := 'F_VN_FillContainerExp_TcVnVector4_SINT_GUID_C28E3CA9_61C1_B75C_67B9_F30C6C109F3A'}
	(* Partially fill the container with the specified value. Only possible for containers with basic elements. (expert function) *)
	FUNCTION F_VN_FillContainerExp_TcVnVector4_SINT : HRESULT
	VAR_INPUT
		ipContainer	:	ITcVnContainer;	(* Container with basic elements *)
	END_VAR
	VAR_IN_OUT
		aValue	:	TcVnVector4_SINT;	(* Value to set the container elements *)
	END_VAR
	VAR_INPUT
		nStartIdx	:	ULINT;	(* Start index *)
		nCount	:	ULINT;	(* Number of elements to set *)
		hrPrev	:	HRESULT;	(* HRESULT indicating the result of previous operations (If SUCCEEDED(hrPrev) equals false, no operation is executed.) *)
	END_VAR

END_FUNCTION

// Functions/Basic Container Operations/F_VN_FillContainerExp/F_VN_FillContainerExp_TcVnVector4_UINT

	{attribute 'TcIecLibraryType'}
	{attribute 'external_name' := 'F_VN_FillContainerExp_TcVnVector4_UINT_GUID_9B232262_EB66_B2E9_4011_444EF75A1E96'}
	(* Partially fill the container with the specified value. Only possible for containers with basic elements. (expert function) *)
	FUNCTION F_VN_FillContainerExp_TcVnVector4_UINT : HRESULT
	VAR_INPUT
		ipContainer	:	ITcVnContainer;	(* Container with basic elements *)
	END_VAR
	VAR_IN_OUT
		aValue	:	TcVnVector4_UINT;	(* Value to set the container elements *)
	END_VAR
	VAR_INPUT
		nStartIdx	:	ULINT;	(* Start index *)
		nCount	:	ULINT;	(* Number of elements to set *)
		hrPrev	:	HRESULT;	(* HRESULT indicating the result of previous operations (If SUCCEEDED(hrPrev) equals false, no operation is executed.) *)
	END_VAR

END_FUNCTION

// Functions/Basic Container Operations/F_VN_FillContainerExp/F_VN_FillContainerExp_TcVnVector4_USINT

	{attribute 'TcIecLibraryType'}
	{attribute 'external_name' := 'F_VN_FillContainerExp_TcVnVector4_USINT_GUID_7CD764AF_E215_BF86_5E3A_97AE5735C37A'}
	(* Partially fill the container with the specified value. Only possible for containers with basic elements. (expert function) *)
	FUNCTION F_VN_FillContainerExp_TcVnVector4_USINT : HRESULT
	VAR_INPUT
		ipContainer	:	ITcVnContainer;	(* Container with basic elements *)
	END_VAR
	VAR_IN_OUT
		aValue	:	TcVnVector4_USINT;	(* Value to set the container elements *)
	END_VAR
	VAR_INPUT
		nStartIdx	:	ULINT;	(* Start index *)
		nCount	:	ULINT;	(* Number of elements to set *)
		hrPrev	:	HRESULT;	(* HRESULT indicating the result of previous operations (If SUCCEEDED(hrPrev) equals false, no operation is executed.) *)
	END_VAR

END_FUNCTION

// Functions/Basic Container Operations/F_VN_FillContainerExp/F_VN_FillContainerExp_UDINT

	{attribute 'TcIecLibraryType'}
	{attribute 'external_name' := 'F_VN_FillContainerExp_UDINT_GUID_35A8E24A_7131_B69C_4943_ACA427C882EA'}
	(* Partially fill the container with the specified value. Only possible for containers with basic elements. (expert function) *)
	FUNCTION F_VN_FillContainerExp_UDINT : HRESULT
	VAR_INPUT
		ipContainer	:	ITcVnContainer;	(* Container with basic elements *)
		nValue	:	UDINT;	(* Value to set the container elements *)
		nStartIdx	:	ULINT;	(* Start index *)
		nCount	:	ULINT;	(* Number of elements to set *)
		hrPrev	:	HRESULT;	(* HRESULT indicating the result of previous operations (If SUCCEEDED(hrPrev) equals false, no operation is executed.) *)
	END_VAR

END_FUNCTION

// Functions/Basic Container Operations/F_VN_FillContainerExp/F_VN_FillContainerExp_UINT

	{attribute 'TcIecLibraryType'}
	{attribute 'external_name' := 'F_VN_FillContainerExp_UINT_GUID_B204A94A_62CF_BADF_7B32_6265D6128185'}
	(* Partially fill the container with the specified value. Only possible for containers with basic elements. (expert function) *)
	FUNCTION F_VN_FillContainerExp_UINT : HRESULT
	VAR_INPUT
		ipContainer	:	ITcVnContainer;	(* Container with basic elements *)
		nValue	:	UINT;	(* Value to set the container elements *)
		nStartIdx	:	ULINT;	(* Start index *)
		nCount	:	ULINT;	(* Number of elements to set *)
		hrPrev	:	HRESULT;	(* HRESULT indicating the result of previous operations (If SUCCEEDED(hrPrev) equals false, no operation is executed.) *)
	END_VAR

END_FUNCTION

// Functions/Basic Container Operations/F_VN_FillContainerExp/F_VN_FillContainerExp_ULINT

	{attribute 'TcIecLibraryType'}
	{attribute 'external_name' := 'F_VN_FillContainerExp_ULINT_GUID_15766B65_3171_B7CF_4898_E019CE5D8C70'}
	(* Partially fill the container with the specified value. Only possible for containers with basic elements. (expert function) *)
	FUNCTION F_VN_FillContainerExp_ULINT : HRESULT
	VAR_INPUT
		ipContainer	:	ITcVnContainer;	(* Container with basic elements *)
		nValue	:	ULINT;	(* Value to set the container elements *)
		nStartIdx	:	ULINT;	(* Start index *)
		nCount	:	ULINT;	(* Number of elements to set *)
		hrPrev	:	HRESULT;	(* HRESULT indicating the result of previous operations (If SUCCEEDED(hrPrev) equals false, no operation is executed.) *)
	END_VAR

END_FUNCTION

// Functions/Basic Container Operations/F_VN_FillContainerExp/F_VN_FillContainerExp_USINT

	{attribute 'TcIecLibraryType'}
	{attribute 'external_name' := 'F_VN_FillContainerExp_USINT_GUID_AACF610B_D842_B80E_50B3_58CDB9F871BA'}
	(* Partially fill the container with the specified value. Only possible for containers with basic elements. (expert function) *)
	FUNCTION F_VN_FillContainerExp_USINT : HRESULT
	VAR_INPUT
		ipContainer	:	ITcVnContainer;	(* Container with basic elements *)
		nValue	:	USINT;	(* Value to set the container elements *)
		nStartIdx	:	ULINT;	(* Start index *)
		nCount	:	ULINT;	(* Number of elements to set *)
		hrPrev	:	HRESULT;	(* HRESULT indicating the result of previous operations (If SUCCEEDED(hrPrev) equals false, no operation is executed.) *)
	END_VAR

END_FUNCTION

// Functions/Basic Container Operations/F_VN_GetAt/F_VN_GetAt_ITcVnContainer

	{attribute 'TcIecLibraryType'}
	{attribute 'external_name' := 'F_VN_GetAt_ITcVnContainer_GUID_F07ECC5F_236B_B5CC_53F7_0424E1B24844'}
	(* Gets the ITcVnContainer element at the specified index of the source container. (Alternatively use interface method .GetAt.) *)
	FUNCTION F_VN_GetAt_ITcVnContainer : HRESULT
	VAR_INPUT
		ipSrcContainer	:	ITcVnContainer;	(* Container with ITcVnContainer elements *)
		ipDestContainer	:	REFERENCE TO ITcVnContainer;	(* Returns the container at the specified index *)
		nIndex	:	ULINT;	(* Index of the requested element *)
		hrPrev	:	HRESULT;	(* HRESULT indicating the result of previous operations (If SUCCEEDED(hrPrev) equals false, no operation is executed.) *)
	END_VAR

END_FUNCTION

// Functions/Basic Container Operations/F_VN_GetAt/F_VN_GetAt_DINT

	{attribute 'TcIecLibraryType'}
	{attribute 'external_name' := 'F_VN_GetAt_DINT_GUID_27D843C5_EBC1_B2D9_78CC_224DD0868EC9'}
	(* Gets the DINT element at the specified index of the container. *)
	FUNCTION F_VN_GetAt_DINT : HRESULT
	VAR_INPUT
		ipContainer	:	ITcVnContainer;	(* Container with DINT elements *)
	END_VAR
	VAR_IN_OUT
		nElement	:	DINT;	(* Returns the element at the specified index *)
	END_VAR
	VAR_INPUT
		nIndex	:	ULINT;	(* Index of the requested element *)
		hrPrev	:	HRESULT;	(* HRESULT indicating the result of previous operations (If SUCCEEDED(hrPrev) equals false, no operation is executed.) *)
	END_VAR

END_FUNCTION

// Functions/Basic Container Operations/F_VN_GetAt/F_VN_GetAt_INT

	{attribute 'TcIecLibraryType'}
	{attribute 'external_name' := 'F_VN_GetAt_INT_GUID_6FA238AB_D13E_B870_5077_8E696A1C078C'}
	(* Gets the INT element at the specified index of the container. *)
	FUNCTION F_VN_GetAt_INT : HRESULT
	VAR_INPUT
		ipContainer	:	ITcVnContainer;	(* Container with INT elements *)
	END_VAR
	VAR_IN_OUT
		nElement	:	INT;	(* Returns the element at the specified index *)
	END_VAR
	VAR_INPUT
		nIndex	:	ULINT;	(* Index of the requested element *)
		hrPrev	:	HRESULT;	(* HRESULT indicating the result of previous operations (If SUCCEEDED(hrPrev) equals false, no operation is executed.) *)
	END_VAR

END_FUNCTION

// Functions/Basic Container Operations/F_VN_GetAt/F_VN_GetAt_ITcVnImage

	{attribute 'TcIecLibraryType'}
	{attribute 'external_name' := 'F_VN_GetAt_ITcVnImage_GUID_68B70C94_079D_B08B_561D_DEBD9AB42794'}
	(* Gets the ITcVnImage element at the specified index of the container. *)
	FUNCTION F_VN_GetAt_ITcVnImage : HRESULT
	VAR_INPUT
		ipContainer	:	ITcVnContainer;	(* Container with ITcVnImage elements *)
		ipElement	:	REFERENCE TO ITcVnImage;	(* Returns the element at the specified index *)
		nIndex	:	ULINT;	(* Index of the requested element *)
		hrPrev	:	HRESULT;	(* HRESULT indicating the result of previous operations (If SUCCEEDED(hrPrev) equals false, no operation is executed.) *)
	END_VAR

END_FUNCTION

// Functions/Basic Container Operations/F_VN_GetAt/F_VN_GetAt_LREAL

